LIN {X 0,Y 395.403,Z 549.53,A -85,B 0,C 180,E1 10502.646,E2 10502.646} C_VEL
LIN {X 0,Y 395.709,Z 549.53,A -85,B 0,C 180,E1 10509.858,E2 10509.858} C_VEL
LIN {X 0,Y 395.987,Z 549.53,A -85,B 0,C 180,E1 10516.739,E2 10516.739} C_VEL
LIN {X 0,Y 396.289,Z 549.53,A -85,B 0,C 180,E1 10523.419,E2 10523.419} C_VEL
LIN {X 0,Y 396.65,Z 549.53,A -85,B 0,C 180,E1 10530.001,E2 10530.001} C_VEL
LIN {X 0,Y 396.335,Z 549.53,A -85,B 0,C 180,E1 10536.637,E2 10536.637} C_VEL
LIN {X 0,Y 395.986,Z 549.53,A -85,B 0,C 180,E1 10543.263,E2 10543.263} C_VEL
LIN {X 0,Y 395.756,Z 549.53,A -85,B 0,C 180,E1 10550.141,E2 10550.141} C_VEL
LIN {X 0,Y 395.466,Z 549.53,A -85,B 0,C 180,E1 10557.351,E2 10557.351} C_VEL
LIN {X 0,Y 395.491,Z 550.097,A -85,B 0,C 180,E1 10559.532,E2 10559.532} C_VEL
LIN {X 0,Y 412.664,Z 588.423,A -85,B 0,C 180,E1 10563.55,E2 10563.55} C_VEL
LIN {X 0,Y 423.549,Z 621.01,A -85,B 0,C 180,E1 10567.103,E2 10567.103} C_VEL
LIN {X 0,Y 418.173,Z 655.721,A -85,B 0,C 180,E1 10570.02,E2 10570.02} C_VEL
LIN {X 0,Y 412.096,Z 688.084,A -85,B 0,C 180,E1 10573.717,E2 10573.717} C_VEL
LIN {X 0,Y 406.338,Z 717.384,A -85,B 0,C 180,E1 10578.3,E2 10578.3} C_VEL
LIN {X 0,Y 402.093,Z 739.295,A -85,B 0,C 180,E1 10582.948,E2 10582.948} C_VEL
LIN {X 0,Y 399.09,Z 757.709,A -85,B 0,C 180,E1 10588.375,E2 10588.375} C_VEL
LIN {X 0,Y 397.658,Z 769.165,A -85,B 0,C 180,E1 10593.25,E2 10593.25} C_VEL
LIN {X 0,Y 396.853,Z 777.225,A -85,B 0,C 180,E1 10598.856,E2 10598.856} C_VEL
LIN {X 0,Y 396.449,Z 780.25,A -85,B 0,C 180,E1 10604.49,E2 10604.49} C_VEL
LIN {X 0,Y 396.674,Z 779.113,A -85,B 0,C 180,E1 10608.994,E2 10608.994} C_VEL
LIN {X 0,Y 397.418,Z 773.339,A -85,B 0,C 180,E1 10614.53,E2 10614.53} C_VEL
LIN {X 0,Y 398.697,Z 762.63,A -85,B 0,C 180,E1 10619.995,E2 10619.995} C_VEL
LIN {X 0,Y 401.47,Z 745.337,A -85,B 0,C 180,E1 10625.677,E2 10625.677} C_VEL
LIN {X 0,Y 405.434,Z 724.606,A -85,B 0,C 180,E1 10630.485,E2 10630.485} C_VEL
LIN {X 0,Y 410.682,Z 698.334,A -85,B 0,C 180,E1 10634.951,E2 10634.951} C_VEL
LIN {X 0,Y 416.116,Z 669.777,A -85,B 0,C 180,E1 10638.554,E2 10638.554} C_VEL
LIN {X 0,Y 421.808,Z 635.983,A -85,B 0,C 180,E1 10641.689,E2 10641.689} C_VEL
LIN {X 0,Y 423.501,Z 620.063,A -85,B 0,C 180,E1 10642.925,E2 10642.925} C_VEL
LIN {X 0,Y 412.42,Z 583.384,A -85,B 0,C 180,E1 10646.95,E2 10646.95} C_VEL
LIN {X 0,Y 402.327,Z 561.945,A -85,B 0,C 180,E1 10649.923,E2 10649.923} C_VEL
LIN {X 0,Y 397.745,Z 555.179,A -85,B 0,C 180,E1 10651.335,E2 10651.335} C_VEL
LIN {X 0,Y 395.279,Z 549.53,A -85,B 0,C 180,E1 10652.574,E2 10652.574} C_VEL
LIN {X 0,Y 395.232,Z 549.53,A -85,B 0,C 180,E1 10659.988,E2 10659.988} C_VEL
LIN {X 0,Y 395.279,Z 549.906,A -85,B 0,C 180,E1 10661.254,E2 10661.254} C_VEL
LIN {X 0,Y 397.807,Z 555.344,A -85,B 0,C 180,E1 10662.27,E2 10662.27} C_VEL
LIN {X 0,Y 400.263,Z 559.059,A -85,B 0,C 180,E1 10663.025,E2 10663.025} C_VEL
LIN {X 0,Y 407.693,Z 571.468,A -85,B 0,C 180,E1 10664.926,E2 10664.926} C_VEL
LIN {X 0,Y 418.785,Z 595.422,A -85,B 0,C 180,E1 10667.342,E2 10667.342} C_VEL
LIN {X 0,Y 427.601,Z 621.106,A -85,B 0,C 180,E1 10669.337,E2 10669.337} C_VEL
LIN {X 0,Y 422.708,Z 664.153,A -85,B 0,C 180,E1 10671.265,E2 10671.265} C_VEL
LIN {X 0,Y 417.375,Z 703.599,A -85,B 0,C 180,E1 10673.921,E2 10673.921} C_VEL
LIN {X 0,Y 412.016,Z 738.43,A -85,B 0,C 180,E1 10677.157,E2 10677.157} C_VEL
LIN {X 0,Y 406.992,Z 769.935,A -85,B 0,C 180,E1 10681.077,E2 10681.077} C_VEL
LIN {X 0,Y 404.873,Z 783.295,A -85,B 0,C 180,E1 10683.114,E2 10683.114} C_VEL
LIN {X 0,Y 399.318,Z 794.258,A -85,B 0,C 180,E1 10684.901,E2 10684.901} C_VEL
LIN {X 0,Y 393.912,Z 804.392,A -85,B 0,C 180,E1 10686.826,E2 10686.826} C_VEL
LIN {X 0,Y 391.203,Z 824.838,A -85,B 0,C 180,E1 10691.962,E2 10691.962} C_VEL
LIN {X 0,Y 389.705,Z 839.343,A -85,B 0,C 180,E1 10697.09,E2 10697.09} C_VEL
LIN {X 0,Y 389.124,Z 849,A -85,B 0,C 180,E1 10702.358,E2 10702.358} C_VEL
LIN {X 0,Y 389.002,Z 853.738,A -85,B 0,C 180,E1 10707.768,E2 10707.768} C_VEL
LIN {X 0,Y 389.053,Z 853.851,A -85,B 0,C 180,E1 10712.229,E2 10712.229} C_VEL
LIN {X 0,Y 389.114,Z 849.446,A -85,B 0,C 180,E1 10717.639,E2 10717.639} C_VEL
LIN {X 0,Y 389.754,Z 840.25,A -85,B 0,C 180,E1 10722.906,E2 10722.906} C_VEL
LIN {X 0,Y 391.432,Z 824.911,A -85,B 0,C 180,E1 10728.513,E2 10728.513} C_VEL
LIN {X 0,Y 394.656,Z 803.613,A -85,B 0,C 180,E1 10733.964,E2 10733.964} C_VEL
LIN {X 0,Y 399.5,Z 777.225,A -85,B 0,C 180,E1 10738.894,E2 10738.894} C_VEL
LIN {X 0,Y 405.396,Z 746.474,A -85,B 0,C 180,E1 10743.154,E2 10743.154} C_VEL
LIN {X 0,Y 411.499,Z 713.376,A -85,B 0,C 180,E1 10746.554,E2 10746.554} C_VEL
LIN {X 0,Y 417.568,Z 675.206,A -85,B 0,C 180,E1 10749.384,E2 10749.384} C_VEL
LIN {X 0,Y 422.691,Z 635.88,A -85,B 0,C 180,E1 10751.334,E2 10751.334} C_VEL
LIN {X 0,Y 423.319,Z 622.141,A -85,B 0,C 180,E1 10751.901,E2 10751.901} C_VEL
LIN {X 0,Y 406.224,Z 585.26,A -85,B 0,C 180,E1 10754.989,E2 10754.989} C_VEL
LIN {X 0,Y 387.369,Z 550.77,A -85,B 0,C 180,E1 10758.29,E2 10758.29} C_VEL
LIN {X 0,Y 387.271,Z 549.53,A -85,B 0,C 180,E1 10758.354,E2 10758.354} C_VEL
LIN {X 0,Y 387.319,Z 549.53,A -85,B 0,C 180,E1 10765.174,E2 10765.174} C_VEL
LIN {X 0,Y 387.507,Z 549.53,A -85,B 0,C 180,E1 10772.046,E2 10772.046} C_VEL
LIN {X 0,Y 387.75,Z 549.53,A -85,B 0,C 180,E1 10779.574,E2 10779.574} C_VEL
LIN {X 0,Y 388.026,Z 549.53,A -85,B 0,C 180,E1 10786.466,E2 10786.466} C_VEL
LIN {X 0,Y 388.335,Z 549.53,A -85,B 0,C 180,E1 10793.288,E2 10793.288} C_VEL
LIN {X 0,Y 388.676,Z 549.53,A -85,B 0,C 180,E1 10800.005,E2 10800.005} C_VEL
LIN {X 0,Y 388.415,Z 549.53,A -85,B 0,C 180,E1 10806.72,E2 10806.72} C_VEL
LIN {X 0,Y 388.038,Z 549.53,A -85,B 0,C 180,E1 10813.544,E2 10813.544} C_VEL
LIN {X 0,Y 387.754,Z 549.53,A -85,B 0,C 180,E1 10820.579,E2 10820.579} C_VEL
LIN {X 0,Y 387.504,Z 549.53,A -85,B 0,C 180,E1 10827.965,E2 10827.965} C_VEL
LIN {X 0,Y 387.251,Z 549.53,A -85,B 0,C 180,E1 10835.911,E2 10835.911} C_VEL
LIN {X 0,Y 387.182,Z 549.53,A -85,B 0,C 180,E1 10842.015,E2 10842.015} C_VEL
LIN {X 0,Y 387.146,Z 549.53,A -85,B 0,C 180,E1 10848.331,E2 10848.331} C_VEL
LIN {X 0,Y 387.311,Z 549.53,A -85,B 0,C 180,E1 10855.184,E2 10855.184} C_VEL
LIN {X 0,Y 387.502,Z 549.53,A -85,B 0,C 180,E1 10862.04,E2 10862.04} C_VEL
LIN {X 0,Y 387.775,Z 549.53,A -85,B 0,C 180,E1 10869.576,E2 10869.576} C_VEL
LIN {X 0,Y 388.059,Z 549.53,A -85,B 0,C 180,E1 10876.463,E2 10876.463} C_VEL
LIN {X 0,Y 388.366,Z 549.53,A -85,B 0,C 180,E1 10883.284,E2 10883.284} C_VEL
LIN {X 0,Y 388.755,Z 549.53,A -85,B 0,C 180,E1 10890.001,E2 10890.001} C_VEL
LIN {X 0,Y 388.445,Z 549.53,A -85,B 0,C 180,E1 10896.716,E2 10896.716} C_VEL
LIN {X 0,Y 388.059,Z 549.53,A -85,B 0,C 180,E1 10903.539,E2 10903.539} C_VEL
LIN {X 0,Y 387.784,Z 549.53,A -85,B 0,C 180,E1 10910.574,E2 10910.574} C_VEL
LIN {X 0,Y 387.559,Z 549.53,A -85,B 0,C 180,E1 10918.428,E2 10918.428} C_VEL
LIN {X 0,Y 406.176,Z 591.509,A -85,B 0,C 180,E1 10923.037,E2 10923.037} C_VEL
LIN {X 0,Y 416.831,Z 624.119,A -85,B 0,C 180,E1 10926.704,E2 10926.704} C_VEL
LIN {X 0,Y 410.701,Z 660.444,A -85,B 0,C 180,E1 10929.862,E2 10929.862} C_VEL
LIN {X 0,Y 404.48,Z 691.718,A -85,B 0,C 180,E1 10933.61,E2 10933.61} C_VEL
LIN {X 0,Y 398.9,Z 718.643,A -85,B 0,C 180,E1 10937.967,E2 10937.967} C_VEL
LIN {X 0,Y 394.176,Z 741.909,A -85,B 0,C 180,E1 10943.082,E2 10943.082} C_VEL
LIN {X 0,Y 391.259,Z 759.109,A -85,B 0,C 180,E1 10948.36,E2 10948.36} C_VEL
LIN {X 0,Y 389.678,Z 771.52,A -85,B 0,C 180,E1 10953.988,E2 10953.988} C_VEL
LIN {X 0,Y 388.911,Z 778.598,A -85,B 0,C 180,E1 10959.485,E2 10959.485} C_VEL
LIN {X 0,Y 388.566,Z 780.931,A -85,B 0,C 180,E1 10964.167,E2 10964.167} C_VEL
LIN {X 0,Y 388.787,Z 780.069,A -85,B 0,C 180,E1 10968.767,E2 10968.767} C_VEL
LIN {X 0,Y 389.581,Z 774.519,A -85,B 0,C 180,E1 10974.42,E2 10974.42} C_VEL
LIN {X 0,Y 390.871,Z 764.073,A -85,B 0,C 180,E1 10979.995,E2 10979.995} C_VEL
LIN {X 0,Y 393.623,Z 748.116,A -85,B 0,C 180,E1 10985.513,E2 10985.513} C_VEL
LIN {X 0,Y 397.902,Z 726.736,A -85,B 0,C 180,E1 10990.685,E2 10990.685} C_VEL
LIN {X 0,Y 403.366,Z 700.882,A -85,B 0,C 180,E1 10995.228,E2 10995.228} C_VEL
LIN {X 0,Y 409.287,Z 671.34,A -85,B 0,C 180,E1 10999.06,E2 10999.06} C_VEL
LIN {X 0,Y 415.229,Z 638,A -85,B 0,C 180,E1 11002.224,E2 11002.224} C_VEL
LIN {X 0,Y 417.094,Z 623.357,A -85,B 0,C 180,E1 11003.371,E2 11003.371} C_VEL
LIN {X 0,Y 406.806,Z 587.316,A -85,B 0,C 180,E1 11007.54,E2 11007.54} C_VEL
LIN {X 0,Y 397.957,Z 567.705,A -85,B 0,C 180,E1 11010.474,E2 11010.474} C_VEL
LIN {X 0,Y 391.388,Z 556.424,A -85,B 0,C 180,E1 11013.09,E2 11013.09} C_VEL
LIN {X 0,Y 387.503,Z 551.323,A -85,B 0,C 180,E1 11016.395,E2 11016.395} C_VEL
LIN {X 0,Y 388.184,Z 553.232,A -85,B 0,C 180,E1 11018.548,E2 11018.548} C_VEL
LIN {X 0,Y 392.347,Z 557.901,A -85,B 0,C 180,E1 11020.909,E2 11020.909} C_VEL
LIN {X 0,Y 399.347,Z 569.21,A -85,B 0,C 180,E1 11023.307,E2 11023.307} C_VEL
LIN {X 0,Y 409.854,Z 590.808,A -85,B 0,C 180,E1 11025.985,E2 11025.985} C_VEL
LIN {X 0,Y 420.921,Z 623.838,A -85,B 0,C 180,E1 11028.792,E2 11028.792} C_VEL
LIN {X 0,Y 415.851,Z 665.501,A -85,B 0,C 180,E1 11030.756,E2 11030.756} C_VEL
LIN {X 0,Y 410.134,Z 705.08,A -85,B 0,C 180,E1 11033.516,E2 11033.516} C_VEL
LIN {X 0,Y 404.212,Z 742.136,A -85,B 0,C 180,E1 11037.117,E2 11037.117} C_VEL
LIN {X 0,Y 398.711,Z 774.627,A -85,B 0,C 180,E1 11041.416,E2 11041.416} C_VEL
LIN {X 0,Y 394.369,Z 801.581,A -85,B 0,C 180,E1 11046.226,E2 11046.226} C_VEL
LIN {X 0,Y 393.912,Z 804.392,A -85,B 0,C 180,E1 11046.826,E2 11046.826} C_VEL
LIN {X 0,Y 392.024,Z 809.183,A -85,B 0,C 180,E1 11047.859,E2 11047.859} C_VEL
LIN {X 0,Y 383.939,Z 820.98,A -85,B 0,C 180,E1 11050.755,E2 11050.755} C_VEL
LIN {X 0,Y 383.723,Z 821.96,A -85,B 0,C 180,E1 11051.047,E2 11051.047} C_VEL
LIN {X 0,Y 381.996,Z 837.115,A -85,B 0,C 180,E1 11056.241,E2 11056.241} C_VEL
LIN {X 0,Y 381.365,Z 846.181,A -85,B 0,C 180,E1 11060.861,E2 11060.861} C_VEL
LIN {X 0,Y 381.15,Z 851.589,A -85,B 0,C 180,E1 11065.442,E2 11065.442} C_VEL
LIN {X 0,Y 381.219,Z 853.512,A -85,B 0,C 180,E1 11069.999,E2 11069.999} C_VEL
LIN {X 0,Y 381.128,Z 850.973,A -85,B 0,C 180,E1 11075.699,E2 11075.699} C_VEL
LIN {X 0,Y 381.581,Z 843.003,A -85,B 0,C 180,E1 11081.442,E2 11081.442} C_VEL
LIN {X 0,Y 383.006,Z 829.207,A -85,B 0,C 180,E1 11087.245,E2 11087.245} C_VEL
LIN {X 0,Y 386.095,Z 808.653,A -85,B 0,C 180,E1 11093.087,E2 11093.087} C_VEL
LIN {X 0,Y 390.87,Z 782.989,A -85,B 0,C 180,E1 11098.317,E2 11098.317} C_VEL
LIN {X 0,Y 396.66,Z 754.143,A -85,B 0,C 180,E1 11102.678,E2 11102.678} C_VEL
LIN {X 0,Y 403.169,Z 720.965,A -85,B 0,C 180,E1 11106.401,E2 11106.401} C_VEL
LIN {X 0,Y 409.328,Z 685.638,A -85,B 0,C 180,E1 11109.303,E2 11109.303} C_VEL
LIN {X 0,Y 414.945,Z 647.471,A -85,B 0,C 180,E1 11111.474,E2 11111.474} C_VEL
LIN {X 0,Y 416.878,Z 624.907,A -85,B 0,C 180,E1 11112.446,E2 11112.446} C_VEL
LIN {X 0,Y 399.707,Z 587.708,A -85,B 0,C 180,E1 11115.694,E2 11115.694} C_VEL
LIN {X 0,Y 379.261,Z 550.017,A -85,B 0,C 180,E1 11119.416,E2 11119.416} C_VEL
LIN {X 0,Y 379.445,Z 549.53,A -85,B 0,C 180,E1 11126.922,E2 11126.922} C_VEL
LIN {X 0,Y 379.598,Z 549.53,A -85,B 0,C 180,E1 11133.982,E2 11133.982} C_VEL
LIN {X 0,Y 379.883,Z 549.53,A -85,B 0,C 180,E1 11141.412,E2 11141.412} C_VEL
LIN {X 0,Y 380.175,Z 549.53,A -85,B 0,C 180,E1 11148.519,E2 11148.519} C_VEL
LIN {X 0,Y 380.544,Z 549.53,A -85,B 0,C 180,E1 11155.441,E2 11155.441} C_VEL
LIN {X 0,Y 380.805,Z 549.53,A -85,B 0,C 180,E1 11162.283,E2 11162.283} C_VEL
LIN {X 0,Y 380.312,Z 549.53,A -85,B 0,C 180,E1 11169.168,E2 11169.168} C_VEL
LIN {X 0,Y 379.993,Z 549.53,A -85,B 0,C 180,E1 11176.2,E2 11176.2} C_VEL
LIN {X 0,Y 379.691,Z 549.53,A -85,B 0,C 180,E1 11183.505,E2 11183.505} C_VEL
LIN {X 0,Y 379.522,Z 549.53,A -85,B 0,C 180,E1 11188.64,E2 11188.64} C_VEL
LIN {X 0,Y 379.353,Z 549.53,A -85,B 0,C 180,E1 11193.975,E2 11193.975} C_VEL
LIN {X 0,Y 379.199,Z 549.53,A -85,B 0,C 180,E1 11200.658,E2 11200.658} C_VEL
LIN {X 0,Y 379.163,Z 549.53,A -85,B 0,C 180,E1 11207.248,E2 11207.248} C_VEL
LIN {X 0,Y 379.259,Z 549.53,A -85,B 0,C 180,E1 11213.215,E2 11213.215} C_VEL
LIN {X 0,Y 379.424,Z 549.53,A -85,B 0,C 180,E1 11218.752,E2 11218.752} C_VEL
LIN {X 0,Y 379.651,Z 549.53,A -85,B 0,C 180,E1 11226.498,E2 11226.498} C_VEL
LIN {X 0,Y 380.009,Z 549.53,A -85,B 0,C 180,E1 11233.806,E2 11233.806} C_VEL
LIN {X 0,Y 380.345,Z 549.53,A -85,B 0,C 180,E1 11240.839,E2 11240.839} C_VEL
LIN {X 0,Y 380.768,Z 549.53,A -85,B 0,C 180,E1 11247.722,E2 11247.722} C_VEL
LIN {X 0,Y 380.544,Z 549.53,A -85,B 0,C 180,E1 11254.565,E2 11254.565} C_VEL
LIN {X 0,Y 380.178,Z 549.53,A -85,B 0,C 180,E1 11261.487,E2 11261.487} C_VEL
LIN {X 0,Y 379.933,Z 549.53,A -85,B 0,C 180,E1 11268.592,E2 11268.592} C_VEL
LIN {X 0,Y 379.667,Z 549.53,A -85,B 0,C 180,E1 11276.02,E2 11276.02} C_VEL
LIN {X 0,Y 379.62,Z 549.767,A -85,B 0,C 180,E1 11277.463,E2 11277.463} C_VEL
LIN {X 0,Y 396.65,Z 587.157,A -85,B 0,C 180,E1 11281.66,E2 11281.66} C_VEL
LIN {X 0,Y 407.431,Z 617.515,A -85,B 0,C 180,E1 11285.154,E2 11285.154} C_VEL
LIN {X 0,Y 409.836,Z 628.295,A -85,B 0,C 180,E1 11286.371,E2 11286.371} C_VEL
LIN {X 0,Y 403.587,Z 662.712,A -85,B 0,C 180,E1 11289.471,E2 11289.471} C_VEL
LIN {X 0,Y 397.063,Z 694.134,A -85,B 0,C 180,E1 11293.345,E2 11293.345} C_VEL
LIN {X 0,Y 391.503,Z 719.773,A -85,B 0,C 180,E1 11297.596,E2 11297.596} C_VEL
LIN {X 0,Y 386.689,Z 742.384,A -85,B 0,C 180,E1 11302.652,E2 11302.652} C_VEL
LIN {X 0,Y 383.785,Z 758.729,A -85,B 0,C 180,E1 11307.669,E2 11307.669} C_VEL
LIN {X 0,Y 381.954,Z 771.588,A -85,B 0,C 180,E1 11313.422,E2 11313.422} C_VEL
LIN {X 0,Y 381.129,Z 779.042,A -85,B 0,C 180,E1 11319.047,E2 11319.047} C_VEL
LIN {X 0,Y 380.695,Z 781.607,A -85,B 0,C 180,E1 11323.831,E2 11323.831} C_VEL
LIN {X 0,Y 380.905,Z 780.952,A -85,B 0,C 180,E1 11328.532,E2 11328.532} C_VEL
LIN {X 0,Y 381.725,Z 775.68,A -85,B 0,C 180,E1 11334.305,E2 11334.305} C_VEL
LIN {X 0,Y 383.074,Z 765.499,A -85,B 0,C 180,E1 11339.995,E2 11339.995} C_VEL
LIN {X 0,Y 385.914,Z 749.858,A -85,B 0,C 180,E1 11345.624,E2 11345.624} C_VEL
LIN {X 0,Y 390.657,Z 727.583,A -85,B 0,C 180,E1 11351.169,E2 11351.169} C_VEL
LIN {X 0,Y 396.455,Z 701.727,A -85,B 0,C 180,E1 11355.784,E2 11355.784} C_VEL
LIN {X 0,Y 402.57,Z 672.766,A -85,B 0,C 180,E1 11359.607,E2 11359.607} C_VEL
LIN {X 0,Y 408.78,Z 639.82,A -85,B 0,C 180,E1 11362.801,E2 11362.801} C_VEL
LIN {X 0,Y 410.607,Z 625.996,A -85,B 0,C 180,E1 11363.924,E2 11363.924} C_VEL
LIN {X 0,Y 401.362,Z 591.182,A -85,B 0,C 180,E1 11368.161,E2 11368.161} C_VEL
LIN {X 0,Y 393.451,Z 572.822,A -85,B 0,C 180,E1 11371.155,E2 11371.155} C_VEL
LIN {X 0,Y 388.4,Z 563.472,A -85,B 0,C 180,E1 11373.572,E2 11373.572} C_VEL
LIN {X 0,Y 385.702,Z 558.895,A -85,B 0,C 180,E1 11376.643,E2 11376.643} C_VEL
LIN {X 0,Y 387.625,Z 562.694,A -85,B 0,C 180,E1 11379.483,E2 11379.483} C_VEL
LIN {X 0,Y 389.867,Z 565.725,A -85,B 0,C 180,E1 11380.663,E2 11380.663} C_VEL
LIN {X 0,Y 396.008,Z 576.315,A -85,B 0,C 180,E1 11382.965,E2 11382.965} C_VEL
LIN {X 0,Y 405.521,Z 597.346,A -85,B 0,C 180,E1 11385.653,E2 11385.653} C_VEL
LIN {X 0,Y 414.457,Z 626.276,A -85,B 0,C 180,E1 11388.219,E2 11388.219} C_VEL
LIN {X 0,Y 408.852,Z 668.458,A -85,B 0,C 180,E1 11390.314,E2 11390.314} C_VEL
LIN {X 0,Y 402.463,Z 709.436,A -85,B 0,C 180,E1 11393.333,E2 11393.333} C_VEL
LIN {X 0,Y 396.386,Z 745.076,A -85,B 0,C 180,E1 11397.003,E2 11397.003} C_VEL
LIN {X 0,Y 391.015,Z 775.388,A -85,B 0,C 180,E1 11401.188,E2 11401.188} C_VEL
LIN {X 0,Y 386.608,Z 801.678,A -85,B 0,C 180,E1 11406.025,E2 11406.025} C_VEL
LIN {X 0,Y 383.723,Z 821.96,A -85,B 0,C 180,E1 11411.047,E2 11411.047} C_VEL
LIN {X 0,Y 380.541,Z 827.599,A -85,B 0,C 180,E1 11412.77,E2 11412.77} C_VEL
LIN {X 0,Y 374.405,Z 834.833,A -85,B 0,C 180,E1 11415.415,E2 11415.415} C_VEL
LIN {X 0,Y 374.233,Z 835.617,A -85,B 0,C 180,E1 11415.728,E2 11415.728} C_VEL
LIN {X 0,Y 373.5,Z 845.344,A -85,B 0,C 180,E1 11420.667,E2 11420.667} C_VEL
LIN {X 0,Y 373.272,Z 850.797,A -85,B 0,C 180,E1 11425.346,E2 11425.346} C_VEL
LIN {X 0,Y 373.37,Z 852.773,A -85,B 0,C 180,E1 11429.999,E2 11429.999} C_VEL
LIN {X 0,Y 373.266,Z 850.397,A -85,B 0,C 180,E1 11435.627,E2 11435.627} C_VEL
LIN {X 0,Y 373.676,Z 843.277,A -85,B 0,C 180,E1 11441.095,E2 11441.095} C_VEL
LIN {X 0,Y 374.794,Z 831.64,A -85,B 0,C 180,E1 11446.425,E2 11446.425} C_VEL
LIN {X 0,Y 377.464,Z 813.611,A -85,B 0,C 180,E1 11452.074,E2 11452.074} C_VEL
LIN {X 0,Y 381.896,Z 790.449,A -85,B 0,C 180,E1 11457.317,E2 11457.317} C_VEL
LIN {X 0,Y 387.58,Z 762.592,A -85,B 0,C 180,E1 11461.992,E2 11461.992} C_VEL
LIN {X 0,Y 393.997,Z 731.725,A -85,B 0,C 180,E1 11465.862,E2 11465.862} C_VEL
LIN {X 0,Y 400.746,Z 697.058,A -85,B 0,C 180,E1 11469.062,E2 11469.062} C_VEL
LIN {X 0,Y 406.674,Z 660.675,A -85,B 0,C 180,E1 11471.452,E2 11471.452} C_VEL
LIN {X 0,Y 410.203,Z 627.23,A -85,B 0,C 180,E1 11473.036,E2 11473.036} C_VEL
LIN {X 0,Y 393.747,Z 591.126,A -85,B 0,C 180,E1 11476.303,E2 11476.303} C_VEL
LIN {X 0,Y 371.419,Z 550.834,A -85,B 0,C 180,E1 11480.496,E2 11480.496} C_VEL
LIN {X 0,Y 371.29,Z 549.53,A -85,B 0,C 180,E1 11480.785,E2 11480.785} C_VEL
LIN {X 0,Y 371.497,Z 549.53,A -85,B 0,C 180,E1 11488.013,E2 11488.013} C_VEL
LIN {X 0,Y 371.67,Z 549.53,A -85,B 0,C 180,E1 11495.966,E2 11495.966} C_VEL
LIN {X 0,Y 372.061,Z 549.53,A -85,B 0,C 180,E1 11503.455,E2 11503.455} C_VEL
LIN {X 0,Y 372.378,Z 549.53,A -85,B 0,C 180,E1 11510.645,E2 11510.645} C_VEL
LIN {X 0,Y 372.782,Z 549.53,A -85,B 0,C 180,E1 11517.677,E2 11517.677} C_VEL
LIN {X 0,Y 372.888,Z 549.53,A -85,B 0,C 180,E1 11522.332,E2 11522.332} C_VEL
LIN {X 0,Y 372.373,Z 549.53,A -85,B 0,C 180,E1 11529.365,E2 11529.365} C_VEL
LIN {X 0,Y 372.071,Z 549.53,A -85,B 0,C 180,E1 11536.555,E2 11536.555} C_VEL
LIN {X 0,Y 371.714,Z 549.53,A -85,B 0,C 180,E1 11544.041,E2 11544.041} C_VEL
LIN {X 0,Y 371.492,Z 549.53,A -85,B 0,C 180,E1 11551.145,E2 11551.145} C_VEL
LIN {X 0,Y 371.263,Z 549.53,A -85,B 0,C 180,E1 11557.719,E2 11557.719} C_VEL
LIN {X 0,Y 371.274,Z 549.53,A -85,B 0,C 180,E1 11563.894,E2 11563.894} C_VEL
LIN {X 0,Y 371.256,Z 549.53,A -85,B 0,C 180,E1 11570.798,E2 11570.798} C_VEL
LIN {X 0,Y 371.498,Z 549.53,A -85,B 0,C 180,E1 11578.008,E2 11578.008} C_VEL
LIN {X 0,Y 371.68,Z 549.53,A -85,B 0,C 180,E1 11585.962,E2 11585.962} C_VEL
LIN {X 0,Y 372.085,Z 549.53,A -85,B 0,C 180,E1 11593.452,E2 11593.452} C_VEL
LIN {X 0,Y 372.407,Z 549.53,A -85,B 0,C 180,E1 11600.642,E2 11600.642} C_VEL
LIN {X 0,Y 372.859,Z 549.53,A -85,B 0,C 180,E1 11607.674,E2 11607.674} C_VEL
LIN {X 0,Y 372.895,Z 549.53,A -85,B 0,C 180,E1 11612.328,E2 11612.328} C_VEL
LIN {X 0,Y 372.394,Z 549.53,A -85,B 0,C 180,E1 11619.361,E2 11619.361} C_VEL
LIN {X 0,Y 372.101,Z 549.53,A -85,B 0,C 180,E1 11626.55,E2 11626.55} C_VEL
LIN {X 0,Y 371.741,Z 549.53,A -85,B 0,C 180,E1 11634.036,E2 11634.036} C_VEL
LIN {X 0,Y 371.743,Z 549.53,A -85,B 0,C 180,E1 11636.351,E2 11636.351} C_VEL
LIN {X 0,Y 378.606,Z 564.621,A -85,B 0,C 180,E1 11638.047,E2 11638.047} C_VEL
LIN {X 0,Y 393.249,Z 597.892,A -85,B 0,C 180,E1 11642.009,E2 11642.009} C_VEL
LIN {X 0,Y 403.104,Z 629.27,A -85,B 0,C 180,E1 11645.756,E2 11645.756} C_VEL
LIN {X 0,Y 396.611,Z 664.345,A -85,B 0,C 180,E1 11648.995,E2 11648.995} C_VEL
LIN {X 0,Y 390.002,Z 694.877,A -85,B 0,C 180,E1 11652.829,E2 11652.829} C_VEL
LIN {X 0,Y 383.799,Z 722.207,A -85,B 0,C 180,E1 11657.478,E2 11657.478} C_VEL
LIN {X 0,Y 378.993,Z 743.931,A -85,B 0,C 180,E1 11662.5,E2 11662.5} C_VEL
LIN {X 0,Y 375.887,Z 760.449,A -85,B 0,C 180,E1 11667.768,E2 11667.768} C_VEL
LIN {X 0,Y 374.094,Z 772.834,A -85,B 0,C 180,E1 11673.559,E2 11673.559} C_VEL
LIN {X 0,Y 373.297,Z 779.703,A -85,B 0,C 180,E1 11678.888,E2 11678.888} C_VEL
LIN {X 0,Y 372.831,Z 782.285,A -85,B 0,C 180,E1 11683.48,E2 11683.48} C_VEL
LIN {X 0,Y 373.012,Z 781.841,A -85,B 0,C 180,E1 11688.286,E2 11688.286} C_VEL
LIN {X 0,Y 373.875,Z 776.824,A -85,B 0,C 180,E1 11694.201,E2 11694.201} C_VEL
LIN {X 0,Y 375.255,Z 766.962,A -85,B 0,C 180,E1 11699.995,E2 11699.995} C_VEL
LIN {X 0,Y 378.203,Z 751.625,A -85,B 0,C 180,E1 11705.739,E2 11705.739} C_VEL
LIN {X 0,Y 382.884,Z 731.039,A -85,B 0,C 180,E1 11711.11,E2 11711.11} C_VEL
LIN {X 0,Y 389.218,Z 704.427,A -85,B 0,C 180,E1 11716.086,E2 11716.086} C_VEL
LIN {X 0,Y 395.834,Z 674.708,A -85,B 0,C 180,E1 11720.131,E2 11720.131} C_VEL
LIN {X 0,Y 402.412,Z 641.64,A -85,B 0,C 180,E1 11723.411,E2 11723.411} C_VEL
LIN {X 0,Y 404.066,Z 628.441,A -85,B 0,C 180,E1 11724.548,E2 11724.548} C_VEL
LIN {X 0,Y 395.849,Z 594.745,A -85,B 0,C 180,E1 11728.865,E2 11728.865} C_VEL
LIN {X 0,Y 388.533,Z 576.11,A -85,B 0,C 180,E1 11732.212,E2 11732.212} C_VEL
LIN {X 0,Y 385.348,Z 570.356,A -85,B 0,C 180,E1 11734.106,E2 11734.106} C_VEL
LIN {X 0,Y 383.822,Z 566.965,A -85,B 0,C 180,E1 11736.271,E2 11736.271} C_VEL
LIN {X 0,Y 384.156,Z 568.14,A -85,B 0,C 180,E1 11738.086,E2 11738.086} C_VEL
LIN {X 0,Y 387.053,Z 572.668,A -85,B 0,C 180,E1 11740.267,E2 11740.267} C_VEL
LIN {X 0,Y 392.786,Z 583.519,A -85,B 0,C 180,E1 11742.643,E2 11742.643} C_VEL
LIN {X 0,Y 401.104,Z 603.996,A -85,B 0,C 180,E1 11745.317,E2 11745.317} C_VEL
LIN {X 0,Y 407.947,Z 629.582,A -85,B 0,C 180,E1 11747.645,E2 11747.645} C_VEL
LIN {X 0,Y 401.622,Z 673.297,A -85,B 0,C 180,E1 11749.982,E2 11749.982} C_VEL
LIN {X 0,Y 394.93,Z 712.853,A -85,B 0,C 180,E1 11753.08,E2 11753.08} C_VEL
LIN {X 0,Y 388.777,Z 746.941,A -85,B 0,C 180,E1 11756.753,E2 11756.753} C_VEL
LIN {X 0,Y 383.024,Z 778.032,A -85,B 0,C 180,E1 11761.245,E2 11761.245} C_VEL
LIN {X 0,Y 378.352,Z 804.531,A -85,B 0,C 180,E1 11766.41,E2 11766.41} C_VEL
LIN {X 0,Y 375.476,Z 824.667,A -85,B 0,C 180,E1 11771.788,E2 11771.788} C_VEL
LIN {X 0,Y 374.233,Z 835.617,A -85,B 0,C 180,E1 11775.728,E2 11775.728} C_VEL
LIN {X 0,Y 371.371,Z 839.752,A -85,B 0,C 180,E1 11777.594,E2 11777.594} C_VEL
LIN {X 0,Y 365.604,Z 845,A -85,B 0,C 180,E1 11780.807,E2 11780.807} C_VEL
LIN {X 0,Y 365.394,Z 850.021,A -85,B 0,C 180,E1 11785.245,E2 11785.245} C_VEL
LIN {X 0,Y 365.522,Z 852.031,A -85,B 0,C 180,E1 11789.999,E2 11789.999} C_VEL
LIN {X 0,Y 365.354,Z 850.408,A -85,B 0,C 180,E1 11794.753,E2 11794.753} C_VEL
LIN {X 0,Y 365.762,Z 843.535,A -85,B 0,C 180,E1 11800.735,E2 11800.735} C_VEL
LIN {X 0,Y 366.845,Z 832.426,A -85,B 0,C 180,E1 11806.175,E2 11806.175} C_VEL
LIN {X 0,Y 369.54,Z 814.548,A -85,B 0,C 180,E1 11812.063,E2 11812.063} C_VEL
LIN {X 0,Y 374.177,Z 791.131,A -85,B 0,C 180,E1 11817.55,E2 11817.55} C_VEL
LIN {X 0,Y 380.12,Z 763.354,A -85,B 0,C 180,E1 11822.358,E2 11822.358} C_VEL
LIN {X 0,Y 386.911,Z 732.115,A -85,B 0,C 180,E1 11826.374,E2 11826.374} C_VEL
LIN {X 0,Y 394.173,Z 695.949,A -85,B 0,C 180,E1 11829.755,E2 11829.755} C_VEL
LIN {X 0,Y 400.543,Z 658.231,A -85,B 0,C 180,E1 11832.231,E2 11832.231} C_VEL
LIN {X 0,Y 403.786,Z 630.204,A -85,B 0,C 180,E1 11833.571,E2 11833.571} C_VEL
LIN {X 0,Y 388.137,Z 595.327,A -85,B 0,C 180,E1 11836.861,E2 11836.861} C_VEL
LIN {X 0,Y 363.449,Z 550.644,A -85,B 0,C 180,E1 11841.682,E2 11841.682} C_VEL
LIN {X 0,Y 363.353,Z 549.53,A -85,B 0,C 180,E1 11841.877,E2 11841.877} C_VEL
LIN {X 0,Y 363.469,Z 549.53,A -85,B 0,C 180,E1 11847.219,E2 11847.219} C_VEL
LIN {X 0,Y 363.624,Z 549.53,A -85,B 0,C 180,E1 11852.747,E2 11852.747} C_VEL
LIN {X 0,Y 363.984,Z 549.53,A -85,B 0,C 180,E1 11860.568,E2 11860.568} C_VEL
LIN {X 0,Y 364.315,Z 549.53,A -85,B 0,C 180,E1 11868.012,E2 11868.012} C_VEL
LIN {X 0,Y 364.727,Z 549.53,A -85,B 0,C 180,E1 11875.243,E2 11875.243} C_VEL
LIN {X 0,Y 364.972,Z 549.53,A -85,B 0,C 180,E1 11882.382,E2 11882.382} C_VEL
LIN {X 0,Y 364.432,Z 549.53,A -85,B 0,C 180,E1 11889.571,E2 11889.571} C_VEL
LIN {X 0,Y 364.12,Z 549.53,A -85,B 0,C 180,E1 11896.99,E2 11896.99} C_VEL
LIN {X 0,Y 363.758,Z 549.53,A -85,B 0,C 180,E1 11904.602,E2 11904.602} C_VEL
LIN {X 0,Y 363.605,Z 549.53,A -85,B 0,C 180,E1 11909.984,E2 11909.984} C_VEL
LIN {X 0,Y 363.376,Z 549.53,A -85,B 0,C 180,E1 11917.66,E2 11917.66} C_VEL
LIN {X 0,Y 363.318,Z 549.53,A -85,B 0,C 180,E1 11924.893,E2 11924.893} C_VEL
LIN {X 0,Y 363.366,Z 549.53,A -85,B 0,C 180,E1 11932.35,E2 11932.35} C_VEL
LIN {X 0,Y 363.613,Z 549.53,A -85,B 0,C 180,E1 11940.023,E2 11940.023} C_VEL
LIN {X 0,Y 363.819,Z 549.53,A -85,B 0,C 180,E1 11948.005,E2 11948.005} C_VEL
LIN {X 0,Y 364.218,Z 549.53,A -85,B 0,C 180,E1 11955.558,E2 11955.558} C_VEL
LIN {X 0,Y 364.605,Z 549.53,A -85,B 0,C 180,E1 11962.845,E2 11962.845} C_VEL
LIN {X 0,Y 365.051,Z 549.53,A -85,B 0,C 180,E1 11970.001,E2 11970.001} C_VEL
LIN {X 0,Y 364.692,Z 549.53,A -85,B 0,C 180,E1 11977.156,E2 11977.156} C_VEL
LIN {X 0,Y 364.222,Z 549.53,A -85,B 0,C 180,E1 11984.444,E2 11984.444} C_VEL
LIN {X 0,Y 363.868,Z 549.53,A -85,B 0,C 180,E1 11991.994,E2 11991.994} C_VEL
LIN {X 0,Y 363.786,Z 549.797,A -85,B 0,C 180,E1 11995.232,E2 11995.232} C_VEL
LIN {X 0,Y 373.547,Z 570.156,A -85,B 0,C 180,E1 11997.676,E2 11997.676} C_VEL
LIN {X 0,Y 388.204,Z 605.005,A -85,B 0,C 180,E1 12001.952,E2 12001.952} C_VEL
LIN {X 0,Y 396.284,Z 631.972,A -85,B 0,C 180,E1 12005.302,E2 12005.302} C_VEL
LIN {X 0,Y 389.491,Z 666.717,A -85,B 0,C 180,E1 12008.59,E2 12008.59} C_VEL
LIN {X 0,Y 382.588,Z 697.257,A -85,B 0,C 180,E1 12012.541,E2 12012.541} C_VEL
LIN {X 0,Y 376.309,Z 723.715,A -85,B 0,C 180,E1 12017.173,E2 12017.173} C_VEL
LIN {X 0,Y 371.351,Z 745.268,A -85,B 0,C 180,E1 12022.291,E2 12022.291} C_VEL
LIN {X 0,Y 368.103,Z 761.66,A -85,B 0,C 180,E1 12027.671,E2 12027.671} C_VEL
LIN {X 0,Y 366.229,Z 773.925,A -85,B 0,C 180,E1 12033.609,E2 12033.609} C_VEL
LIN {X 0,Y 365.303,Z 781.03,A -85,B 0,C 180,E1 12039.595,E2 12039.595} C_VEL
LIN {X 0,Y 364.98,Z 783.235,A -85,B 0,C 180,E1 12045.583,E2 12045.583} C_VEL
LIN {X 0,Y 365.548,Z 780.502,A -85,B 0,C 180,E1 12051.66,E2 12051.66} C_VEL
LIN {X 0,Y 366.728,Z 772.905,A -85,B 0,C 180,E1 12057.629,E2 12057.629} C_VEL
LIN {X 0,Y 369.079,Z 760.143,A -85,B 0,C 180,E1 12063.523,E2 12063.523} C_VEL
LIN {X 0,Y 373.297,Z 741.432,A -85,B 0,C 180,E1 12069.332,E2 12069.332} C_VEL
LIN {X 0,Y 379.13,Z 718.206,A -85,B 0,C 180,E1 12074.448,E2 12074.448} C_VEL
LIN {X 0,Y 385.871,Z 690.699,A -85,B 0,C 180,E1 12078.882,E2 12078.882} C_VEL
LIN {X 0,Y 393.145,Z 658.726,A -85,B 0,C 180,E1 12082.645,E2 12082.645} C_VEL
LIN {X 0,Y 397.868,Z 631.854,A -85,B 0,C 180,E1 12085.078,E2 12085.078} C_VEL
LIN {X 0,Y 390.753,Z 599.088,A -85,B 0,C 180,E1 12089.493,E2 12089.493} C_VEL
LIN {X 0,Y 384.866,Z 582.333,A -85,B 0,C 180,E1 12092.751,E2 12092.751} C_VEL
LIN {X 0,Y 382.538,Z 577.334,A -85,B 0,C 180,E1 12094.587,E2 12094.587} C_VEL
LIN {X 0,Y 381.866,Z 574.457,A -85,B 0,C 180,E1 12097.072,E2 12097.072} C_VEL
LIN {X 0,Y 384.391,Z 579.833,A -85,B 0,C 180,E1 12099.918,E2 12099.918} C_VEL
LIN {X 0,Y 389.565,Z 590.854,A -85,B 0,C 180,E1 12102.399,E2 12102.399} C_VEL
LIN {X 0,Y 397.24,Z 612.814,A -85,B 0,C 180,E1 12105.217,E2 12105.217} C_VEL
LIN {X 0,Y 401.72,Z 631.423,A -85,B 0,C 180,E1 12106.992,E2 12106.992} C_VEL
LIN {X 0,Y 395.099,Z 673.808,A -85,B 0,C 180,E1 12109.347,E2 12109.347} C_VEL
LIN {X 0,Y 388.119,Z 712.679,A -85,B 0,C 180,E1 12112.471,E2 12112.471} C_VEL
LIN {X 0,Y 381.377,Z 748.024,A -85,B 0,C 180,E1 12116.384,E2 12116.384} C_VEL
LIN {X 0,Y 375.295,Z 779.149,A -85,B 0,C 180,E1 12121.044,E2 12121.044} C_VEL
LIN {X 0,Y 370.469,Z 805.258,A -85,B 0,C 180,E1 12126.336,E2 12126.336} C_VEL
LIN {X 0,Y 367.616,Z 824.588,A -85,B 0,C 180,E1 12131.687,E2 12131.687} C_VEL
LIN {X 0,Y 366.056,Z 838.399,A -85,B 0,C 180,E1 12137.091,E2 12137.091} C_VEL
LIN {X 0,Y 365.604,Z 845,A -85,B 0,C 180,E1 12140.807,E2 12140.807} C_VEL
LIN {X 0,Y 364.225,Z 846.756,A -85,B 0,C 180,E1 12142.136,E2 12142.136} C_VEL
LIN {X 0,Y 357.475,Z 849.916,A -85,B 0,C 180,E1 12146.087,E2 12146.087} C_VEL
LIN {X 0,Y 357.468,Z 849.861,A -85,B 0,C 180,E1 12146.174,E2 12146.174} C_VEL
LIN {X 0,Y 357.666,Z 851.288,A -85,B 0,C 180,E1 12149.999,E2 12149.999} C_VEL
LIN {X 0,Y 357.501,Z 849.671,A -85,B 0,C 180,E1 12154.858,E2 12154.858} C_VEL
LIN {X 0,Y 357.883,Z 842.769,A -85,B 0,C 180,E1 12160.974,E2 12160.974} C_VEL
LIN {X 0,Y 359.04,Z 831.603,A -85,B 0,C 180,E1 12166.537,E2 12166.537} C_VEL
LIN {X 0,Y 362.075,Z 813.067,A -85,B 0,C 180,E1 12172.687,E2 12172.687} C_VEL
LIN {X 0,Y 367.032,Z 789.176,A -85,B 0,C 180,E1 12178.319,E2 12178.319} C_VEL
LIN {X 0,Y 373.292,Z 761.333,A -85,B 0,C 180,E1 12183.144,E2 12183.144} C_VEL
LIN {X 0,Y 380.612,Z 728.825,A -85,B 0,C 180,E1 12187.298,E2 12187.298} C_VEL
LIN {X 0,Y 388.275,Z 691.783,A -85,B 0,C 180,E1 12190.714,E2 12190.714} C_VEL
LIN {X 0,Y 395.109,Z 652.042,A -85,B 0,C 180,E1 12193.227,E2 12193.227} C_VEL
LIN {X 0,Y 397.026,Z 632.119,A -85,B 0,C 180,E1 12194.212,E2 12194.212} C_VEL
LIN {X 0,Y 380.793,Z 596.117,A -85,B 0,C 180,E1 12197.77,E2 12197.77} C_VEL
LIN {X 0,Y 355.523,Z 550.708,A -85,B 0,C 180,E1 12202.9,E2 12202.9} C_VEL
LIN {X 0,Y 355.437,Z 549.53,A -85,B 0,C 180,E1 12203.144,E2 12203.144} C_VEL
LIN {X 0,Y 355.595,Z 549.53,A -85,B 0,C 180,E1 12209.28,E2 12209.28} C_VEL
LIN {X 0,Y 355.732,Z 549.53,A -85,B 0,C 180,E1 12214.816,E2 12214.816} C_VEL
LIN {X 0,Y 356.171,Z 549.53,A -85,B 0,C 180,E1 12222.694,E2 12222.694} C_VEL
LIN {X 0,Y 356.5,Z 549.53,A -85,B 0,C 180,E1 12230.225,E2 12230.225} C_VEL
LIN {X 0,Y 356.965,Z 549.53,A -85,B 0,C 180,E1 12237.574,E2 12237.574} C_VEL
LIN {X 0,Y 357.084,Z 549.53,A -85,B 0,C 180,E1 12242.435,E2 12242.435} C_VEL
LIN {X 0,Y 356.492,Z 549.53,A -85,B 0,C 180,E1 12249.786,E2 12249.786} C_VEL
LIN {X 0,Y 356.191,Z 549.53,A -85,B 0,C 180,E1 12257.315,E2 12257.315} C_VEL
LIN {X 0,Y 355.763,Z 549.53,A -85,B 0,C 180,E1 12265.192,E2 12265.192} C_VEL
LIN {X 0,Y 355.502,Z 549.53,A -85,B 0,C 180,E1 12271.595,E2 12271.595} C_VEL
LIN {X 0,Y 355.438,Z 549.53,A -85,B 0,C 180,E1 12276.615,E2 12276.615} C_VEL
LIN {X 0,Y 355.316,Z 549.53,A -85,B 0,C 180,E1 12283.582,E2 12283.582} C_VEL
LIN {X 0,Y 355.353,Z 549.53,A -85,B 0,C 180,E1 12290.276,E2 12290.276} C_VEL
LIN {X 0,Y 355.507,Z 549.53,A -85,B 0,C 180,E1 12296.383,E2 12296.383} C_VEL
LIN {X 0,Y 355.714,Z 549.53,A -85,B 0,C 180,E1 12303.369,E2 12303.369} C_VEL
LIN {X 0,Y 356.025,Z 549.53,A -85,B 0,C 180,E1 12310.111,E2 12310.111} C_VEL
LIN {X 0,Y 356.412,Z 549.53,A -85,B 0,C 180,E1 12317.738,E2 12317.738} C_VEL
LIN {X 0,Y 356.932,Z 549.53,A -85,B 0,C 180,E1 12325.134,E2 12325.134} C_VEL
LIN {X 0,Y 357.091,Z 549.53,A -85,B 0,C 180,E1 12332.431,E2 12332.431} C_VEL
LIN {X 0,Y 356.514,Z 549.53,A -85,B 0,C 180,E1 12339.782,E2 12339.782} C_VEL
LIN {X 0,Y 356.213,Z 549.53,A -85,B 0,C 180,E1 12347.31,E2 12347.31} C_VEL
LIN {X 0,Y 355.908,Z 549.614,A -85,B 0,C 180,E1 12354.045,E2 12354.045} C_VEL
LIN {X 0,Y 360.496,Z 559.885,A -85,B 0,C 180,E1 12355.25,E2 12355.25} C_VEL
LIN {X 0,Y 376.506,Z 594.418,A -85,B 0,C 180,E1 12359.679,E2 12359.679} C_VEL
LIN {X 0,Y 387.222,Z 625.776,A -85,B 0,C 180,E1 12363.678,E2 12363.678} C_VEL
LIN {X 0,Y 389.141,Z 636.065,A -85,B 0,C 180,E1 12364.936,E2 12364.936} C_VEL
LIN {X 0,Y 381.862,Z 671.195,A -85,B 0,C 180,E1 12368.413,E2 12368.413} C_VEL
LIN {X 0,Y 374.463,Z 702.631,A -85,B 0,C 180,E1 12372.716,E2 12372.716} C_VEL
LIN {X 0,Y 368.134,Z 728.098,A -85,B 0,C 180,E1 12377.462,E2 12377.462} C_VEL
LIN {X 0,Y 363.141,Z 749.029,A -85,B 0,C 180,E1 12382.773,E2 12382.773} C_VEL
LIN {X 0,Y 359.93,Z 764.863,A -85,B 0,C 180,E1 12388.378,E2 12388.378} C_VEL
LIN {X 0,Y 358.356,Z 775.094,A -85,B 0,C 180,E1 12393.712,E2 12393.712} C_VEL
LIN {X 0,Y 357.532,Z 781.148,A -85,B 0,C 180,E1 12398.696,E2 12398.696} C_VEL
LIN {X 0,Y 357.088,Z 784.019,A -85,B 0,C 180,E1 12405.257,E2 12405.257} C_VEL
LIN {X 0,Y 357.655,Z 781.368,A -85,B 0,C 180,E1 12411.593,E2 12411.593} C_VEL
LIN {X 0,Y 358.898,Z 774.291,A -85,B 0,C 180,E1 12417.577,E2 12417.577} C_VEL
LIN {X 0,Y 361.356,Z 761.85,A -85,B 0,C 180,E1 12423.598,E2 12423.598} C_VEL
LIN {X 0,Y 365.734,Z 743.504,A -85,B 0,C 180,E1 12429.526,E2 12429.526} C_VEL
LIN {X 0,Y 371.791,Z 720.722,A -85,B 0,C 180,E1 12434.74,E2 12434.74} C_VEL
LIN {X 0,Y 378.809,Z 693.808,A -85,B 0,C 180,E1 12439.248,E2 12439.248} C_VEL
LIN {X 0,Y 386.304,Z 662.657,A -85,B 0,C 180,E1 12443.069,E2 12443.069} C_VEL
LIN {X 0,Y 391.739,Z 634.83,A -85,B 0,C 180,E1 12445.693,E2 12445.693} C_VEL
LIN {X 0,Y 385.677,Z 602.731,A -85,B 0,C 180,E1 12450.268,E2 12450.268} C_VEL
LIN {X 0,Y 381.125,Z 587.898,A -85,B 0,C 180,E1 12453.521,E2 12453.521} C_VEL
LIN {X 0,Y 379.718,Z 584.063,A -85,B 0,C 180,E1 12455.194,E2 12455.194} C_VEL
LIN {X 0,Y 379.686,Z 582.416,A -85,B 0,C 180,E1 12457.276,E2 12457.276} C_VEL
LIN {X 0,Y 381.65,Z 587.263,A -85,B 0,C 180,E1 12459.674,E2 12459.674} C_VEL
LIN {X 0,Y 386.123,Z 598.366,A -85,B 0,C 180,E1 12462.13,E2 12462.13} C_VEL
LIN {X 0,Y 392.413,Z 619.195,A -85,B 0,C 180,E1 12464.863,E2 12464.863} C_VEL
LIN {X 0,Y 395.541,Z 633.732,A -85,B 0,C 180,E1 12466.326,E2 12466.326} C_VEL
LIN {X 0,Y 388.422,Z 675.822,A -85,B 0,C 180,E1 12468.779,E2 12468.779} C_VEL
LIN {X 0,Y 380.801,Z 715.747,A -85,B 0,C 180,E1 12472.136,E2 12472.136} C_VEL
LIN {X 0,Y 373.618,Z 750.775,A -85,B 0,C 180,E1 12476.221,E2 12476.221} C_VEL
LIN {X 0,Y 367.375,Z 781.304,A -85,B 0,C 180,E1 12481.035,E2 12481.035} C_VEL
LIN {X 0,Y 362.663,Z 805.632,A -85,B 0,C 180,E1 12486.181,E2 12486.181} C_VEL
LIN {X 0,Y 359.622,Z 825.368,A -85,B 0,C 180,E1 12491.889,E2 12491.889} C_VEL
LIN {X 0,Y 358.038,Z 839.483,A -85,B 0,C 180,E1 12497.792,E2 12497.792} C_VEL
LIN {X 0,Y 357.53,Z 848.083,A -85,B 0,C 180,E1 12503.774,E2 12503.774} C_VEL
LIN {X 0,Y 357.468,Z 849.861,A -85,B 0,C 180,E1 12506.174,E2 12506.174} C_VEL
LIN {X 0,Y 354.982,Z 850.689,A -85,B 0,C 180,E1 12508.243,E2 12508.243} C_VEL
LIN {X 0,Y 349.695,Z 850.283,A -85,B 0,C 180,E1 12511.733,E2 12511.733} C_VEL
LIN {X 0,Y 349.727,Z 846.819,A -85,B 0,C 180,E1 12517.461,E2 12517.461} C_VEL
LIN {X 0,Y 350.374,Z 838.558,A -85,B 0,C 180,E1 12523.23,E2 12523.23} C_VEL
LIN {X 0,Y 352.271,Z 824.092,A -85,B 0,C 180,E1 12529.422,E2 12529.422} C_VEL
LIN {X 0,Y 356.272,Z 803.612,A -85,B 0,C 180,E1 12535.441,E2 12535.441} C_VEL
LIN {X 0,Y 361.971,Z 778.679,A -85,B 0,C 180,E1 12540.741,E2 12540.741} C_VEL
LIN {X 0,Y 369.057,Z 748.957,A -85,B 0,C 180,E1 12545.413,E2 12545.413} C_VEL
LIN {X 0,Y 376.743,Z 715.548,A -85,B 0,C 180,E1 12549.268,E2 12549.268} C_VEL
LIN {X 0,Y 384.266,Z 678.053,A -85,B 0,C 180,E1 12552.368,E2 12552.368} C_VEL
LIN {X 0,Y 390.878,Z 636.641,A -85,B 0,C 180,E1 12554.642,E2 12554.642} C_VEL
LIN {X 0,Y 377.337,Z 604.715,A -85,B 0,C 180,E1 12557.876,E2 12557.876} C_VEL
LIN {X 0,Y 355.332,Z 564.778,A -85,B 0,C 180,E1 12562.429,E2 12562.429} C_VEL
LIN {X 0,Y 347.593,Z 550.248,A -85,B 0,C 180,E1 12564.203,E2 12564.203} C_VEL
LIN {X 0,Y 347.706,Z 549.53,A -85,B 0,C 180,E1 12571.387,E2 12571.387} C_VEL
LIN {X 0,Y 348.05,Z 549.53,A -85,B 0,C 180,E1 12579.64,E2 12579.64} C_VEL
LIN {X 0,Y 348.284,Z 549.53,A -85,B 0,C 180,E1 12584.886,E2 12584.886} C_VEL
LIN {X 0,Y 348.722,Z 549.53,A -85,B 0,C 180,E1 12592.521,E2 12592.521} C_VEL
LIN {X 0,Y 349.183,Z 549.53,A -85,B 0,C 180,E1 12600.005,E2 12600.005} C_VEL
LIN {X 0,Y 348.79,Z 549.53,A -85,B 0,C 180,E1 12607.488,E2 12607.488} C_VEL
LIN {X 0,Y 348.298,Z 549.53,A -85,B 0,C 180,E1 12615.124,E2 12615.124} C_VEL
LIN {X 0,Y 347.9,Z 549.53,A -85,B 0,C 180,E1 12623.064,E2 12623.064} C_VEL
LIN {X 0,Y 347.644,Z 549.53,A -85,B 0,C 180,E1 12629.422,E2 12629.422} C_VEL
LIN {X 0,Y 347.506,Z 549.53,A -85,B 0,C 180,E1 12634.505,E2 12634.505} C_VEL
LIN {X 0,Y 347.349,Z 549.53,A -85,B 0,C 180,E1 12642.184,E2 12642.184} C_VEL
LIN {X 0,Y 347.335,Z 549.53,A -85,B 0,C 180,E1 12649.168,E2 12649.168} C_VEL
LIN {X 0,Y 347.556,Z 549.53,A -85,B 0,C 180,E1 12655.87,E2 12655.87} C_VEL
LIN {X 0,Y 347.697,Z 549.53,A -85,B 0,C 180,E1 12661.381,E2 12661.381} C_VEL
LIN {X 0,Y 348.076,Z 549.53,A -85,B 0,C 180,E1 12669.637,E2 12669.637} C_VEL
LIN {X 0,Y 348.316,Z 549.53,A -85,B 0,C 180,E1 12674.883,E2 12674.883} C_VEL
LIN {X 0,Y 348.752,Z 549.53,A -85,B 0,C 180,E1 12682.518,E2 12682.518} C_VEL
LIN {X 0,Y 349.26,Z 549.53,A -85,B 0,C 180,E1 12690.001,E2 12690.001} C_VEL
LIN {X 0,Y 348.815,Z 549.53,A -85,B 0,C 180,E1 12697.483,E2 12697.483} C_VEL
LIN {X 0,Y 348.321,Z 549.53,A -85,B 0,C 180,E1 12705.119,E2 12705.119} C_VEL
LIN {X 0,Y 348.041,Z 549.885,A -85,B 0,C 180,E1 12712.809,E2 12712.809} C_VEL
LIN {X 0,Y 355.407,Z 565.268,A -85,B 0,C 180,E1 12714.803,E2 12714.803} C_VEL
LIN {X 0,Y 369.988,Z 597.398,A -85,B 0,C 180,E1 12719.076,E2 12719.076} C_VEL
LIN {X 0,Y 380.633,Z 628.98,A -85,B 0,C 180,E1 12723.227,E2 12723.227} C_VEL
LIN {X 0,Y 382.313,Z 638.488,A -85,B 0,C 180,E1 12724.416,E2 12724.416} C_VEL
LIN {X 0,Y 374.672,Z 673.772,A -85,B 0,C 180,E1 12728.02,E2 12728.02} C_VEL
LIN {X 0,Y 367.025,Z 704.823,A -85,B 0,C 180,E1 12732.422,E2 12732.422} C_VEL
LIN {X 0,Y 360.452,Z 730.086,A -85,B 0,C 180,E1 12737.279,E2 12737.279} C_VEL
LIN {X 0,Y 355.22,Z 751.295,A -85,B 0,C 180,E1 12742.881,E2 12742.881} C_VEL
LIN {X 0,Y 351.899,Z 767.328,A -85,B 0,C 180,E1 12748.91,E2 12748.91} C_VEL
LIN {X 0,Y 350.213,Z 778.177,A -85,B 0,C 180,E1 12755.217,E2 12755.217} C_VEL
LIN {X 0,Y 349.533,Z 782.689,A -85,B 0,C 180,E1 12759.72,E2 12759.72} C_VEL
LIN {X 0,Y 349.204,Z 784.785,A -85,B 0,C 180,E1 12764.916,E2 12764.916} C_VEL
LIN {X 0,Y 349.61,Z 783.431,A -85,B 0,C 180,E1 12770.019,E2 12770.019} C_VEL
LIN {X 0,Y 350.789,Z 777.401,A -85,B 0,C 180,E1 12776.283,E2 12776.283} C_VEL
LIN {X 0,Y 353.006,Z 766.357,A -85,B 0,C 180,E1 12782.453,E2 12782.453} C_VEL
LIN {X 0,Y 357.09,Z 749.694,A -85,B 0,C 180,E1 12788.529,E2 12788.529} C_VEL
LIN {X 0,Y 362.958,Z 728.828,A -85,B 0,C 180,E1 12793.873,E2 12793.873} C_VEL
LIN {X 0,Y 370.33,Z 702.49,A -85,B 0,C 180,E1 12798.776,E2 12798.776} C_VEL
LIN {X 0,Y 378.379,Z 671.707,A -85,B 0,C 180,E1 12802.959,E2 12802.959} C_VEL
LIN {X 0,Y 385.777,Z 638.133,A -85,B 0,C 180,E1 12806.303,E2 12806.303} C_VEL
LIN {X 0,Y 381.101,Z 607.713,A -85,B 0,C 180,E1 12810.88,E2 12810.88} C_VEL
LIN {X 0,Y 378.285,Z 595.907,A -85,B 0,C 180,E1 12813.516,E2 12813.516} C_VEL
LIN {X 0,Y 377.129,Z 591.309,A -85,B 0,C 180,E1 12815.472,E2 12815.472} C_VEL
LIN {X 0,Y 377.334,Z 589.747,A -85,B 0,C 180,E1 12816.997,E2 12816.997} C_VEL
LIN {X 0,Y 379.016,Z 595.004,A -85,B 0,C 180,E1 12819.563,E2 12819.563} C_VEL
LIN {X 0,Y 382.688,Z 605.942,A -85,B 0,C 180,E1 12821.914,E2 12821.914} C_VEL
LIN {X 0,Y 387.632,Z 625.782,A -85,B 0,C 180,E1 12824.526,E2 12824.526} C_VEL
LIN {X 0,Y 389.264,Z 637.695,A -85,B 0,C 180,E1 12825.701,E2 12825.701} C_VEL
LIN {X 0,Y 381.433,Z 679.926,A -85,B 0,C 180,E1 12828.334,E2 12828.334} C_VEL
LIN {X 0,Y 373.445,Z 718.829,A -85,B 0,C 180,E1 12831.808,E2 12831.808} C_VEL
LIN {X 0,Y 366.103,Z 752.406,A -85,B 0,C 180,E1 12835.898,E2 12835.898} C_VEL
LIN {X 0,Y 359.778,Z 781.806,A -85,B 0,C 180,E1 12840.71,E2 12840.71} C_VEL
LIN {X 0,Y 354.89,Z 805.748,A -85,B 0,C 180,E1 12845.95,E2 12845.95} C_VEL
LIN {X 0,Y 351.764,Z 825.203,A -85,B 0,C 180,E1 12851.768,E2 12851.768} C_VEL
LIN {X 0,Y 350.199,Z 838.621,A -85,B 0,C 180,E1 12857.515,E2 12857.515} C_VEL
LIN {X 0,Y 349.767,Z 846.102,A -85,B 0,C 180,E1 12862.537,E2 12862.537} C_VEL
LIN {X 0,Y 349.708,Z 849.949,A -85,B 0,C 180,E1 12867.518,E2 12867.518} C_VEL
LIN {X 0,Y 349.695,Z 850.283,A -85,B 0,C 180,E1 12871.733,E2 12871.733} C_VEL
LIN {X 0,Y 347.145,Z 849.386,A -85,B 0,C 180,E1 12873.845,E2 12873.845} C_VEL
LIN {X 0,Y 341.86,Z 846.673,A -85,B 0,C 180,E1 12877.012,E2 12877.012} C_VEL
LIN {X 0,Y 341.809,Z 846.299,A -85,B 0,C 180,E1 12877.378,E2 12877.378} C_VEL
LIN {X 0,Y 342.548,Z 837.769,A -85,B 0,C 180,E1 12883.521,E2 12883.521} C_VEL
LIN {X 0,Y 344.611,Z 822.93,A -85,B 0,C 180,E1 12889.959,E2 12889.959} C_VEL
LIN {X 0,Y 348.574,Z 803.623,A -85,B 0,C 180,E1 12895.743,E2 12895.743} C_VEL
LIN {X 0,Y 354.627,Z 778.225,A -85,B 0,C 180,E1 12901.277,E2 12901.277} C_VEL
LIN {X 0,Y 362.045,Z 748.605,A -85,B 0,C 180,E1 12906.016,E2 12906.016} C_VEL
LIN {X 0,Y 370.043,Z 715.103,A -85,B 0,C 180,E1 12909.93,E2 12909.93} C_VEL
LIN {X 0,Y 377.827,Z 677.587,A -85,B 0,C 180,E1 12913.073,E2 12913.073} C_VEL
LIN {X 0,Y 384.105,Z 638.088,A -85,B 0,C 180,E1 12915.332,E2 12915.332} C_VEL
LIN {X 0,Y 368.895,Z 603.213,A -85,B 0,C 180,E1 12919.057,E2 12919.057} C_VEL
LIN {X 0,Y 344.681,Z 559.984,A -85,B 0,C 180,E1 12924.318,E2 12924.318} C_VEL
LIN {X 0,Y 339.694,Z 550.109,A -85,B 0,C 180,E1 12925.547,E2 12925.547} C_VEL
LIN {X 0,Y 339.758,Z 549.53,A -85,B 0,C 180,E1 12933.03,E2 12933.03} C_VEL
LIN {X 0,Y 340.074,Z 549.53,A -85,B 0,C 180,E1 12939.218,E2 12939.218} C_VEL
LIN {X 0,Y 340.51,Z 549.53,A -85,B 0,C 180,E1 12947.16,E2 12947.16} C_VEL
LIN {X 0,Y 340.989,Z 549.53,A -85,B 0,C 180,E1 12954.911,E2 12954.911} C_VEL
LIN {X 0,Y 341.297,Z 549.53,A -85,B 0,C 180,E1 12960.005,E2 12960.005} C_VEL
LIN {X 0,Y 340.848,Z 549.53,A -85,B 0,C 180,E1 12967.663,E2 12967.663} C_VEL
LIN {X 0,Y 340.366,Z 549.53,A -85,B 0,C 180,E1 12975.485,E2 12975.485} C_VEL
LIN {X 0,Y 339.946,Z 549.53,A -85,B 0,C 180,E1 12983.636,E2 12983.636} C_VEL
LIN {X 0,Y 339.747,Z 549.53,A -85,B 0,C 180,E1 12989.36,E2 12989.36} C_VEL
LIN {X 0,Y 339.428,Z 549.53,A -85,B 0,C 180,E1 12996.593,E2 12996.593} C_VEL
LIN {X 0,Y 339.441,Z 549.53,A -85,B 0,C 180,E1 13002.001,E2 13002.001} C_VEL
LIN {X 0,Y 339.418,Z 549.53,A -85,B 0,C 180,E1 13009.324,E2 13009.324} C_VEL
LIN {X 0,Y 339.651,Z 549.53,A -85,B 0,C 180,E1 13017.662,E2 13017.662} C_VEL
LIN {X 0,Y 339.81,Z 549.53,A -85,B 0,C 180,E1 13023.542,E2 13023.542} C_VEL
LIN {X 0,Y 340.26,Z 549.53,A -85,B 0,C 180,E1 13031.853,E2 13031.853} C_VEL
LIN {X 0,Y 340.652,Z 549.53,A -85,B 0,C 180,E1 13039.76,E2 13039.76} C_VEL
LIN {X 0,Y 341.252,Z 549.53,A -85,B 0,C 180,E1 13047.458,E2 13047.458} C_VEL
LIN {X 0,Y 341.268,Z 549.53,A -85,B 0,C 180,E1 13052.544,E2 13052.544} C_VEL
LIN {X 0,Y 340.635,Z 549.53,A -85,B 0,C 180,E1 13060.242,E2 13060.242} C_VEL
LIN {X 0,Y 340.274,Z 549.53,A -85,B 0,C 180,E1 13068.149,E2 13068.149} C_VEL
LIN {X 0,Y 340.102,Z 549.53,A -85,B 0,C 180,E1 13071.462,E2 13071.462} C_VEL
LIN {X 0,Y 344.818,Z 559.895,A -85,B 0,C 180,E1 13072.816,E2 13072.816} C_VEL
LIN {X 0,Y 360.074,Z 591.968,A -85,B 0,C 180,E1 13077.291,E2 13077.291} C_VEL
LIN {X 0,Y 371.295,Z 622.513,A -85,B 0,C 180,E1 13081.464,E2 13081.464} C_VEL
LIN {X 0,Y 375.542,Z 640.454,A -85,B 0,C 180,E1 13083.856,E2 13083.856} C_VEL
LIN {X 0,Y 367.559,Z 675.826,A -85,B 0,C 180,E1 13087.566,E2 13087.566} C_VEL
LIN {X 0,Y 359.746,Z 706.424,A -85,B 0,C 180,E1 13092.013,E2 13092.013} C_VEL
LIN {X 0,Y 353.154,Z 730.752,A -85,B 0,C 180,E1 13096.79,E2 13096.79} C_VEL
LIN {X 0,Y 347.726,Z 751.804,A -85,B 0,C 180,E1 13102.435,E2 13102.435} C_VEL
LIN {X 0,Y 344.369,Z 767.022,A -85,B 0,C 180,E1 13108.152,E2 13108.152} C_VEL
LIN {X 0,Y 342.669,Z 777.179,A -85,B 0,C 180,E1 13113.773,E2 13113.773} C_VEL
LIN {X 0,Y 341.725,Z 783.111,A -85,B 0,C 180,E1 13119.235,E2 13119.235} C_VEL
LIN {X 0,Y 341.311,Z 785.466,A -85,B 0,C 180,E1 13124.559,E2 13124.559} C_VEL
LIN {X 0,Y 341.733,Z 784.442,A -85,B 0,C 180,E1 13129.787,E2 13129.787} C_VEL
LIN {X 0,Y 342.954,Z 778.718,A -85,B 0,C 180,E1 13136.198,E2 13136.198} C_VEL
LIN {X 0,Y 345.26,Z 768.022,A -85,B 0,C 180,E1 13142.508,E2 13142.508} C_VEL
LIN {X 0,Y 349.523,Z 751.733,A -85,B 0,C 180,E1 13148.715,E2 13148.715} C_VEL
LIN {X 0,Y 355.607,Z 731.314,A -85,B 0,C 180,E1 13154.165,E2 13154.165} C_VEL
LIN {X 0,Y 363.288,Z 705.589,A -85,B 0,C 180,E1 13159.154,E2 13159.154} C_VEL
LIN {X 0,Y 371.647,Z 675.621,A -85,B 0,C 180,E1 13163.399,E2 13163.399} C_VEL
LIN {X 0,Y 379.844,Z 640.825,A -85,B 0,C 180,E1 13167.052,E2 13167.052} C_VEL
LIN {X 0,Y 376.695,Z 612.887,A -85,B 0,C 180,E1 13171.494,E2 13171.494} C_VEL
LIN {X 0,Y 374.788,Z 601.068,A -85,B 0,C 180,E1 13174.435,E2 13174.435} C_VEL
LIN {X 0,Y 374.523,Z 598.161,A -85,B 0,C 180,E1 13176.046,E2 13176.046} C_VEL
LIN {X 0,Y 374.859,Z 597.82,A -85,B 0,C 180,E1 13177.283,E2 13177.283} C_VEL
LIN {X 0,Y 376.423,Z 603.306,A -85,B 0,C 180,E1 13179.623,E2 13179.623} C_VEL
LIN {X 0,Y 379.847,Z 617.26,A -85,B 0,C 180,E1 13182.268,E2 13182.268} C_VEL
LIN {X 0,Y 383.699,Z 638.498,A -85,B 0,C 180,E1 13184.884,E2 13184.884} C_VEL
LIN {X 0,Y 375.08,Z 681.11,A -85,B 0,C 180,E1 13187.65,E2 13187.65} C_VEL
LIN {X 0,Y 366.399,Z 720.626,A -85,B 0,C 180,E1 13191.316,E2 13191.316} C_VEL
LIN {X 0,Y 358.439,Z 754.915,A -85,B 0,C 180,E1 13195.679,E2 13195.679} C_VEL
LIN {X 0,Y 351.399,Z 785.635,A -85,B 0,C 180,E1 13201.004,E2 13201.004} C_VEL
LIN {X 0,Y 346.382,Z 810.111,A -85,B 0,C 180,E1 13206.833,E2 13206.833} C_VEL
LIN {X 0,Y 343.46,Z 827.896,A -85,B 0,C 180,E1 13212.688,E2 13212.688} C_VEL
LIN {X 0,Y 342.193,Z 840.017,A -85,B 0,C 180,E1 13218.514,E2 13218.514} C_VEL
LIN {X 0,Y 341.797,Z 846.635,A -85,B 0,C 180,E1 13223.641,E2 13223.641} C_VEL
LIN {X 0,Y 341.967,Z 849.789,A -85,B 0,C 180,E1 13229.999,E2 13229.999} C_VEL
LIN {X 0,Y 341.735,Z 847.278,A -85,B 0,C 180,E1 13236.358,E2 13236.358} C_VEL
LIN {X 0,Y 341.809,Z 846.299,A -85,B 0,C 180,E1 13237.378,E2 13237.378} C_VEL
LIN {X 0,Y 339.492,Z 843.815,A -85,B 0,C 180,E1 13239.506,E2 13239.506} C_VEL
LIN {X 0,Y 334.556,Z 838.935,A -85,B 0,C 180,E1 13242.683,E2 13242.683} C_VEL
LIN {X 0,Y 334.542,Z 838.358,A -85,B 0,C 180,E1 13243.049,E2 13243.049} C_VEL
LIN {X 0,Y 336.438,Z 824.909,A -85,B 0,C 180,E1 13249.352,E2 13249.352} C_VEL
LIN {X 0,Y 340.554,Z 805.084,A -85,B 0,C 180,E1 13255.687,E2 13255.687} C_VEL
LIN {X 0,Y 346.592,Z 780.815,A -85,B 0,C 180,E1 13261.247,E2 13261.247} C_VEL
LIN {X 0,Y 354.412,Z 750.595,A -85,B 0,C 180,E1 13266.296,E2 13266.296} C_VEL
LIN {X 0,Y 362.629,Z 717.507,A -85,B 0,C 180,E1 13270.327,E2 13270.327} C_VEL
LIN {X 0,Y 370.496,Z 681.677,A -85,B 0,C 180,E1 13273.471,E2 13273.471} C_VEL
LIN {X 0,Y 377.594,Z 642.231,A -85,B 0,C 180,E1 13275.831,E2 13275.831} C_VEL
LIN {X 0,Y 366.085,Z 613.314,A -85,B 0,C 180,E1 13278.97,E2 13278.97} C_VEL
LIN {X 0,Y 345.724,Z 575.214,A -85,B 0,C 180,E1 13283.569,E2 13283.569} C_VEL
LIN {X 0,Y 331.847,Z 550.884,A -85,B 0,C 180,E1 13286.919,E2 13286.919} C_VEL
LIN {X 0,Y 331.728,Z 549.53,A -85,B 0,C 180,E1 13287.108,E2 13287.108} C_VEL
LIN {X 0,Y 331.869,Z 549.53,A -85,B 0,C 180,E1 13292.863,E2 13292.863} C_VEL
LIN {X 0,Y 332.25,Z 549.53,A -85,B 0,C 180,E1 13301.404,E2 13301.404} C_VEL
LIN {X 0,Y 332.694,Z 549.53,A -85,B 0,C 180,E1 13309.517,E2 13309.517} C_VEL
LIN {X 0,Y 333.264,Z 549.53,A -85,B 0,C 180,E1 13317.402,E2 13317.402} C_VEL
LIN {X 0,Y 333.347,Z 549.53,A -85,B 0,C 180,E1 13322.609,E2 13322.609} C_VEL
LIN {X 0,Y 332.676,Z 549.53,A -85,B 0,C 180,E1 13330.494,E2 13330.494} C_VEL
LIN {X 0,Y 332.274,Z 549.53,A -85,B 0,C 180,E1 13338.606,E2 13338.606} C_VEL
LIN {X 0,Y 331.876,Z 549.53,A -85,B 0,C 180,E1 13347.148,E2 13347.148} C_VEL
LIN {X 0,Y 331.537,Z 549.53,A -85,B 0,C 180,E1 13354.714,E2 13354.714} C_VEL
LIN {X 0,Y 331.519,Z 549.53,A -85,B 0,C 180,E1 13359.752,E2 13359.752} C_VEL
LIN {X 0,Y 331.466,Z 549.53,A -85,B 0,C 180,E1 13366.964,E2 13366.964} C_VEL
LIN {X 0,Y 331.551,Z 549.53,A -85,B 0,C 180,E1 13373.584,E2 13373.584} C_VEL
LIN {X 0,Y 331.775,Z 549.53,A -85,B 0,C 180,E1 13380.128,E2 13380.128} C_VEL
LIN {X 0,Y 332.104,Z 549.53,A -85,B 0,C 180,E1 13388.611,E2 13388.611} C_VEL
LIN {X 0,Y 332.42,Z 549.53,A -85,B 0,C 180,E1 13394.142,E2 13394.142} C_VEL
LIN {X 0,Y 332.894,Z 549.53,A -85,B 0,C 180,E1 13402.159,E2 13402.159} C_VEL
LIN {X 0,Y 333.47,Z 549.53,A -85,B 0,C 180,E1 13410.001,E2 13410.001} C_VEL
LIN {X 0,Y 332.941,Z 549.53,A -85,B 0,C 180,E1 13417.842,E2 13417.842} C_VEL
LIN {X 0,Y 332.428,Z 549.53,A -85,B 0,C 180,E1 13425.86,E2 13425.86} C_VEL
LIN {X 0,Y 332.226,Z 549.53,A -85,B 0,C 180,E1 13430.081,E2 13430.081} C_VEL
LIN {X 0,Y 334.659,Z 555.175,A -85,B 0,C 180,E1 13430.85,E2 13430.85} C_VEL
LIN {X 0,Y 350.548,Z 587.705,A -85,B 0,C 180,E1 13435.59,E2 13435.59} C_VEL
LIN {X 0,Y 362.782,Z 619.31,A -85,B 0,C 180,E1 13440.055,E2 13440.055} C_VEL
LIN {X 0,Y 368.809,Z 642.287,A -85,B 0,C 180,E1 13443.268,E2 13443.268} C_VEL
LIN {X 0,Y 360.53,Z 677.55,A -85,B 0,C 180,E1 13447.062,E2 13447.062} C_VEL
LIN {X 0,Y 352.669,Z 707.233,A -85,B 0,C 180,E1 13451.46,E2 13451.46} C_VEL
LIN {X 0,Y 345.715,Z 731.965,A -85,B 0,C 180,E1 13456.41,E2 13456.41} C_VEL
LIN {X 0,Y 340.203,Z 752.484,A -85,B 0,C 180,E1 13462.033,E2 13462.033} C_VEL
LIN {X 0,Y 336.53,Z 768.326,A -85,B 0,C 180,E1 13468.156,E2 13468.156} C_VEL
LIN {X 0,Y 334.746,Z 778.544,A -85,B 0,C 180,E1 13474.05,E2 13474.05} C_VEL
LIN {X 0,Y 333.935,Z 783.53,A -85,B 0,C 180,E1 13478.727,E2 13478.727} C_VEL
LIN {X 0,Y 333.435,Z 786.146,A -85,B 0,C 180,E1 13484.185,E2 13484.185} C_VEL
LIN {X 0,Y 333.825,Z 785.453,A -85,B 0,C 180,E1 13489.542,E2 13489.542} C_VEL
LIN {X 0,Y 335.122,Z 780.057,A -85,B 0,C 180,E1 13496.109,E2 13496.109} C_VEL
LIN {X 0,Y 337.498,Z 769.709,A -85,B 0,C 180,E1 13502.566,E2 13502.566} C_VEL
LIN {X 0,Y 341.953,Z 753.83,A -85,B 0,C 180,E1 13508.909,E2 13508.909} C_VEL
LIN {X 0,Y 348.69,Z 732.574,A -85,B 0,C 180,E1 13514.774,E2 13514.774} C_VEL
LIN {X 0,Y 356.794,Z 707.059,A -85,B 0,C 180,E1 13519.839,E2 13519.839} C_VEL
LIN {X 0,Y 365.7,Z 677.113,A -85,B 0,C 180,E1 13524.18,E2 13524.18} C_VEL
LIN {X 0,Y 374.175,Z 644.556,A -85,B 0,C 180,E1 13527.676,E2 13527.676} C_VEL
LIN {X 0,Y 372.379,Z 617.822,A -85,B 0,C 180,E1 13532.185,E2 13532.185} C_VEL
LIN {X 0,Y 371.73,Z 608.092,A -85,B 0,C 180,E1 13534.759,E2 13534.759} C_VEL
LIN {X 0,Y 371.795,Z 606.388,A -85,B 0,C 180,E1 13535.464,E2 13535.464} C_VEL
LIN {X 0,Y 372.21,Z 605.896,A -85,B 0,C 180,E1 13537.594,E2 13537.594} C_VEL
LIN {X 0,Y 373.376,Z 611.468,A -85,B 0,C 180,E1 13539.603,E2 13539.603} C_VEL
LIN {X 0,Y 376.267,Z 627.903,A -85,B 0,C 180,E1 13542.482,E2 13542.482} C_VEL
LIN {X 0,Y 377.614,Z 642.756,A -85,B 0,C 180,E1 13544.216,E2 13544.216} C_VEL
LIN {X 0,Y 368.032,Z 686.369,A -85,B 0,C 180,E1 13547.25,E2 13547.25} C_VEL
LIN {X 0,Y 358.607,Z 725.842,A -85,B 0,C 180,E1 13551.181,E2 13551.181} C_VEL
LIN {X 0,Y 350.241,Z 759.604,A -85,B 0,C 180,E1 13555.806,E2 13555.806} C_VEL
LIN {X 0,Y 343.417,Z 787.673,A -85,B 0,C 180,E1 13560.988,E2 13560.988} C_VEL
LIN {X 0,Y 338.609,Z 810.262,A -85,B 0,C 180,E1 13566.618,E2 13566.618} C_VEL
LIN {X 0,Y 335.72,Z 826.997,A -85,B 0,C 180,E1 13572.276,E2 13572.276} C_VEL
LIN {X 0,Y 334.355,Z 839.185,A -85,B 0,C 180,E1 13578.241,E2 13578.241} C_VEL
LIN {X 0,Y 333.939,Z 845.851,A -85,B 0,C 180,E1 13583.49,E2 13583.49} C_VEL
LIN {X 0,Y 333.976,Z 848.436,A -85,B 0,C 180,E1 13587.401,E2 13587.401} C_VEL
LIN {X 0,Y 334.002,Z 848.664,A -85,B 0,C 180,E1 13592.597,E2 13592.597} C_VEL
LIN {X 0,Y 334.066,Z 843.908,A -85,B 0,C 180,E1 13599.126,E2 13599.126} C_VEL
LIN {X 0,Y 334.542,Z 838.358,A -85,B 0,C 180,E1 13603.049,E2 13603.049} C_VEL
LIN {X 0,Y 332.511,Z 834.535,A -85,B 0,C 180,E1 13605.18,E2 13605.18} C_VEL
LIN {X 0,Y 328.174,Z 827.593,A -85,B 0,C 180,E1 13608.327,E2 13608.327} C_VEL
LIN {X 0,Y 328.234,Z 826.731,A -85,B 0,C 180,E1 13608.683,E2 13608.683} C_VEL
LIN {X 0,Y 331.95,Z 808.676,A -85,B 0,C 180,E1 13614.954,E2 13614.954} C_VEL
LIN {X 0,Y 337.693,Z 786.092,A -85,B 0,C 180,E1 13620.594,E2 13620.594} C_VEL
LIN {X 0,Y 345.065,Z 758.663,A -85,B 0,C 180,E1 13625.65,E2 13625.65} C_VEL
LIN {X 0,Y 353.529,Z 726.739,A -85,B 0,C 180,E1 13629.97,E2 13629.97} C_VEL
LIN {X 0,Y 362.12,Z 690.514,A -85,B 0,C 180,E1 13633.495,E2 13633.495} C_VEL
LIN {X 0,Y 369.923,Z 651.224,A -85,B 0,C 180,E1 13636.116,E2 13636.116} C_VEL
LIN {X 0,Y 370.521,Z 642.196,A -85,B 0,C 180,E1 13636.674,E2 13636.674} C_VEL
LIN {X 0,Y 355.601,Z 607.428,A -85,B 0,C 180,E1 13640.711,E2 13640.711} C_VEL
LIN {X 0,Y 332.444,Z 565.752,A -85,B 0,C 180,E1 13646.198,E2 13646.198} C_VEL
LIN {X 0,Y 324.044,Z 551.312,A -85,B 0,C 180,E1 13648.359,E2 13648.359} C_VEL
LIN {X 0,Y 323.86,Z 549.53,A -85,B 0,C 180,E1 13648.649,E2 13648.649} C_VEL
LIN {X 0,Y 323.955,Z 549.53,A -85,B 0,C 180,E1 13655.132,E2 13655.132} C_VEL
LIN {X 0,Y 324.262,Z 549.53,A -85,B 0,C 180,E1 13660.929,E2 13660.929} C_VEL
LIN {X 0,Y 324.747,Z 549.53,A -85,B 0,C 180,E1 13669.258,E2 13669.258} C_VEL
LIN {X 0,Y 325.347,Z 549.53,A -85,B 0,C 180,E1 13677.338,E2 13677.338} C_VEL
LIN {X 0,Y 325.427,Z 549.53,A -85,B 0,C 180,E1 13682.672,E2 13682.672} C_VEL
LIN {X 0,Y 324.726,Z 549.53,A -85,B 0,C 180,E1 13690.754,E2 13690.754} C_VEL
LIN {X 0,Y 324.472,Z 549.53,A -85,B 0,C 180,E1 13696.264,E2 13696.264} C_VEL
LIN {X 0,Y 324.144,Z 549.53,A -85,B 0,C 180,E1 13701.948,E2 13701.948} C_VEL
LIN {X 0,Y 323.886,Z 549.53,A -85,B 0,C 180,E1 13707.876,E2 13707.876} C_VEL
LIN {X 0,Y 323.628,Z 549.53,A -85,B 0,C 180,E1 13714.159,E2 13714.159} C_VEL
LIN {X 0,Y 323.463,Z 549.53,A -85,B 0,C 180,E1 13721.504,E2 13721.504} C_VEL
LIN {X 0,Y 323.461,Z 549.53,A -85,B 0,C 180,E1 13729.058,E2 13729.058} C_VEL
LIN {X 0,Y 323.642,Z 549.53,A -85,B 0,C 180,E1 13735.85,E2 13735.85} C_VEL
LIN {X 0,Y 323.935,Z 549.53,A -85,B 0,C 180,E1 13742.639,E2 13742.639} C_VEL
LIN {X 0,Y 324.295,Z 549.53,A -85,B 0,C 180,E1 13750.926,E2 13750.926} C_VEL
LIN {X 0,Y 324.774,Z 549.53,A -85,B 0,C 180,E1 13759.254,E2 13759.254} C_VEL
LIN {X 0,Y 325.449,Z 549.53,A -85,B 0,C 180,E1 13767.335,E2 13767.335} C_VEL
LIN {X 0,Y 325.451,Z 549.53,A -85,B 0,C 180,E1 13772.668,E2 13772.668} C_VEL
LIN {X 0,Y 324.748,Z 549.53,A -85,B 0,C 180,E1 13780.749,E2 13780.749} C_VEL
LIN {X 0,Y 324.399,Z 549.644,A -85,B 0,C 180,E1 13788.689,E2 13788.689} C_VEL
LIN {X 0,Y 326.762,Z 555.228,A -85,B 0,C 180,E1 13789.454,E2 13789.454} C_VEL
LIN {X 0,Y 343.025,Z 587.917,A -85,B 0,C 180,E1 13794.445,E2 13794.445} C_VEL
LIN {X 0,Y 355.786,Z 621.083,A -85,B 0,C 180,E1 13799.302,E2 13799.302} C_VEL
LIN {X 0,Y 361.987,Z 643.952,A -85,B 0,C 180,E1 13802.634,E2 13802.634} C_VEL
LIN {X 0,Y 353.648,Z 678.818,A -85,B 0,C 180,E1 13806.479,E2 13806.479} C_VEL
LIN {X 0,Y 345.421,Z 708.68,A -85,B 0,C 180,E1 13811.003,E2 13811.003} C_VEL
LIN {X 0,Y 338.125,Z 733.602,A -85,B 0,C 180,E1 13816.131,E2 13816.131} C_VEL
LIN {X 0,Y 332.333,Z 754.421,A -85,B 0,C 180,E1 13822.039,E2 13822.039} C_VEL
LIN {X 0,Y 328.744,Z 769.353,A -85,B 0,C 180,E1 13828.024,E2 13828.024} C_VEL
LIN {X 0,Y 326.866,Z 779.629,A -85,B 0,C 180,E1 13834.185,E2 13834.185} C_VEL
LIN {X 0,Y 326.156,Z 783.92,A -85,B 0,C 180,E1 13838.194,E2 13838.194} C_VEL
LIN {X 0,Y 325.571,Z 786.809,A -85,B 0,C 180,E1 13843.792,E2 13843.792} C_VEL
LIN {X 0,Y 325.917,Z 786.388,A -85,B 0,C 180,E1 13849.286,E2 13849.286} C_VEL
LIN {X 0,Y 327.267,Z 781.315,A -85,B 0,C 180,E1 13856.015,E2 13856.015} C_VEL
LIN {X 0,Y 330.112,Z 770.047,A -85,B 0,C 180,E1 13863.281,E2 13863.281} C_VEL
LIN {X 0,Y 334.956,Z 754.007,A -85,B 0,C 180,E1 13869.753,E2 13869.753} C_VEL
LIN {X 0,Y 342.237,Z 732.613,A -85,B 0,C 180,E1 13875.716,E2 13875.716} C_VEL
LIN {X 0,Y 350.962,Z 706.952,A -85,B 0,C 180,E1 13880.843,E2 13880.843} C_VEL
LIN {X 0,Y 360.839,Z 675.921,A -85,B 0,C 180,E1 13885.35,E2 13885.35} C_VEL
LIN {X 0,Y 368.628,Z 647.284,A -85,B 0,C 180,E1 13888.514,E2 13888.514} C_VEL
LIN {X 0,Y 368.355,Z 623.7,A -85,B 0,C 180,E1 13892.72,E2 13892.72} C_VEL
LIN {X 0,Y 368.57,Z 615.025,A -85,B 0,C 180,E1 13895.1,E2 13895.1} C_VEL
LIN {X 0,Y 368.764,Z 613.588,A -85,B 0,C 180,E1 13895.8,E2 13895.8} C_VEL
LIN {X 0,Y 369.509,Z 614.088,A -85,B 0,C 180,E1 13897.917,E2 13897.917} C_VEL
LIN {X 0,Y 370.407,Z 622.81,A -85,B 0,C 180,E1 13900.196,E2 13900.196} C_VEL
LIN {X 0,Y 372.424,Z 642.396,A -85,B 0,C 180,E1 13903.15,E2 13903.15} C_VEL
LIN {X 0,Y 361.41,Z 689.729,A -85,B 0,C 180,E1 13906.684,E2 13906.684} C_VEL
LIN {X 0,Y 351.471,Z 728.326,A -85,B 0,C 180,E1 13910.726,E2 13910.726} C_VEL
LIN {X 0,Y 342.393,Z 762.696,A -85,B 0,C 180,E1 13915.679,E2 13915.679} C_VEL
LIN {X 0,Y 335.115,Z 791.471,A -85,B 0,C 180,E1 13921.358,E2 13921.358} C_VEL
LIN {X 0,Y 330.184,Z 813.518,A -85,B 0,C 180,E1 13927.31,E2 13927.31} C_VEL
LIN {X 0,Y 327.354,Z 830.822,A -85,B 0,C 180,E1 13933.887,E2 13933.887} C_VEL
LIN {X 0,Y 326.24,Z 842.235,A -85,B 0,C 180,E1 13940.651,E2 13940.651} C_VEL
LIN {X 0,Y 326.124,Z 847.683,A -85,B 0,C 180,E1 13947.338,E2 13947.338} C_VEL
LIN {X 0,Y 326.146,Z 847.899,A -85,B 0,C 180,E1 13952.66,E2 13952.66} C_VEL
LIN {X 0,Y 326.094,Z 844.489,A -85,B 0,C 180,E1 13958.006,E2 13958.006} C_VEL
LIN {X 0,Y 327.006,Z 835.028,A -85,B 0,C 180,E1 13964.752,E2 13964.752} C_VEL
LIN {X 0,Y 328.234,Z 826.731,A -85,B 0,C 180,E1 13968.683,E2 13968.683} C_VEL
LIN {X 0,Y 326.749,Z 821.571,A -85,B 0,C 180,E1 13970.773,E2 13970.773} C_VEL
LIN {X 0,Y 323.299,Z 812.986,A -85,B 0,C 180,E1 13973.876,E2 13973.876} C_VEL
LIN {X 0,Y 323.438,Z 811.95,A -85,B 0,C 180,E1 13974.22,E2 13974.22} C_VEL
LIN {X 0,Y 329.734,Z 787.788,A -85,B 0,C 180,E1 13980.671,E2 13980.671} C_VEL
LIN {X 0,Y 337.722,Z 759.262,A -85,B 0,C 180,E1 13986.122,E2 13986.122} C_VEL
LIN {X 0,Y 346.378,Z 727.843,A -85,B 0,C 180,E1 13990.486,E2 13990.486} C_VEL
LIN {X 0,Y 355.163,Z 692.258,A -85,B 0,C 180,E1 13994.058,E2 13994.058} C_VEL
LIN {X 0,Y 362.985,Z 654.877,A -85,B 0,C 180,E1 13996.66,E2 13996.66} C_VEL
LIN {X 0,Y 364.171,Z 645.438,A -85,B 0,C 180,E1 13997.229,E2 13997.229} C_VEL
LIN {X 0,Y 349.328,Z 610.374,A -85,B 0,C 180,E1 14001.488,E2 14001.488} C_VEL
LIN {X 0,Y 327.738,Z 571.065,A -85,B 0,C 180,E1 14006.811,E2 14006.811} C_VEL
LIN {X 0,Y 316.036,Z 551.117,A -85,B 0,C 180,E1 14009.958,E2 14009.958} C_VEL
LIN {X 0,Y 315.846,Z 549.53,A -85,B 0,C 180,E1 14010.143,E2 14010.143} C_VEL
LIN {X 0,Y 316.091,Z 549.53,A -85,B 0,C 180,E1 14017.475,E2 14017.475} C_VEL
LIN {X 0,Y 316.47,Z 549.53,A -85,B 0,C 180,E1 14023.325,E2 14023.325} C_VEL
LIN {X 0,Y 316.984,Z 549.53,A -85,B 0,C 180,E1 14031.768,E2 14031.768} C_VEL
LIN {X 0,Y 317.611,Z 549.53,A -85,B 0,C 180,E1 14040.006,E2 14040.006} C_VEL
LIN {X 0,Y 317.232,Z 549.53,A -85,B 0,C 180,E1 14045.483,E2 14045.483} C_VEL
LIN {X 0,Y 316.629,Z 549.53,A -85,B 0,C 180,E1 14053.838,E2 14053.838} C_VEL
LIN {X 0,Y 316.342,Z 549.53,A -85,B 0,C 180,E1 14059.58,E2 14059.58} C_VEL
LIN {X 0,Y 316.034,Z 549.53,A -85,B 0,C 180,E1 14065.548,E2 14065.548} C_VEL
LIN {X 0,Y 315.747,Z 549.53,A -85,B 0,C 180,E1 14071.841,E2 14071.841} C_VEL
LIN {X 0,Y 315.498,Z 549.53,A -85,B 0,C 180,E1 14079.842,E2 14079.842} C_VEL
LIN {X 0,Y 315.472,Z 549.53,A -85,B 0,C 180,E1 14087.787,E2 14087.787} C_VEL
LIN {X 0,Y 315.616,Z 549.53,A -85,B 0,C 180,E1 14094.856,E2 14094.856} C_VEL
LIN {X 0,Y 315.86,Z 549.53,A -85,B 0,C 180,E1 14101.359,E2 14101.359} C_VEL
LIN {X 0,Y 316.111,Z 549.53,A -85,B 0,C 180,E1 14107.471,E2 14107.471} C_VEL
LIN {X 0,Y 316.506,Z 549.53,A -85,B 0,C 180,E1 14113.322,E2 14113.322} C_VEL
LIN {X 0,Y 317.013,Z 549.53,A -85,B 0,C 180,E1 14121.763,E2 14121.763} C_VEL
LIN {X 0,Y 317.704,Z 549.53,A -85,B 0,C 180,E1 14130.001,E2 14130.001} C_VEL
LIN {X 0,Y 317.047,Z 549.53,A -85,B 0,C 180,E1 14138.238,E2 14138.238} C_VEL
LIN {X 0,Y 316.525,Z 549.53,A -85,B 0,C 180,E1 14146.912,E2 14146.912} C_VEL
LIN {X 0,Y 316.917,Z 552.049,A -85,B 0,C 180,E1 14147.384,E2 14147.384} C_VEL
LIN {X 0,Y 333.131,Z 583.206,A -85,B 0,C 180,E1 14152.478,E2 14152.478} C_VEL
LIN {X 0,Y 345.426,Z 613.018,A -85,B 0,C 180,E1 14157.05,E2 14157.05} C_VEL
LIN {X 0,Y 354.342,Z 642.47,A -85,B 0,C 180,E1 14161.491,E2 14161.491} C_VEL
LIN {X 0,Y 354.572,Z 649.402,A -85,B 0,C 180,E1 14162.396,E2 14162.396} C_VEL
LIN {X 0,Y 345.947,Z 683.018,A -85,B 0,C 180,E1 14166.271,E2 14166.271} C_VEL
LIN {X 0,Y 337.308,Z 713.093,A -85,B 0,C 180,E1 14171.061,E2 14171.061} C_VEL
LIN {X 0,Y 329.489,Z 738.88,A -85,B 0,C 180,E1 14176.759,E2 14176.759} C_VEL
LIN {X 0,Y 323.692,Z 759.343,A -85,B 0,C 180,E1 14183.144,E2 14183.144} C_VEL
LIN {X 0,Y 320.291,Z 773.771,A -85,B 0,C 180,E1 14189.692,E2 14189.692} C_VEL
LIN {X 0,Y 318.586,Z 782.827,A -85,B 0,C 180,E1 14196.169,E2 14196.169} C_VEL
LIN {X 0,Y 317.715,Z 787.176,A -85,B 0,C 180,E1 14202.386,E2 14202.386} C_VEL
LIN {X 0,Y 318.009,Z 787.308,A -85,B 0,C 180,E1 14209.016,E2 14209.016} C_VEL
LIN {X 0,Y 319.191,Z 783.546,A -85,B 0,C 180,E1 14214.966,E2 14214.966} C_VEL
LIN {X 0,Y 321.571,Z 774.181,A -85,B 0,C 180,E1 14222.018,E2 14222.018} C_VEL
LIN {X 0,Y 326.203,Z 759.743,A -85,B 0,C 180,E1 14228.67,E2 14228.67} C_VEL
LIN {X 0,Y 333.23,Z 740.25,A -85,B 0,C 180,E1 14234.802,E2 14234.802} C_VEL
LIN {X 0,Y 342.351,Z 715.346,A -85,B 0,C 180,E1 14240.376,E2 14240.376} C_VEL
LIN {X 0,Y 353.188,Z 684.015,A -85,B 0,C 180,E1 14245.378,E2 14245.378} C_VEL
LIN {X 0,Y 363.328,Z 651.513,A -85,B 0,C 180,E1 14249.148,E2 14249.148} C_VEL
LIN {X 0,Y 364.546,Z 628.474,A -85,B 0,C 180,E1 14253.54,E2 14253.54} C_VEL
LIN {X 0,Y 365.47,Z 621.989,A -85,B 0,C 180,E1 14255.443,E2 14255.443} C_VEL
LIN {X 0,Y 366.291,Z 621.054,A -85,B 0,C 180,E1 14257.55,E2 14257.55} C_VEL
LIN {X 0,Y 366.512,Z 629.133,A -85,B 0,C 180,E1 14259.72,E2 14259.72} C_VEL
LIN {X 0,Y 367.205,Z 646.78,A -85,B 0,C 180,E1 14262.474,E2 14262.474} C_VEL
LIN {X 0,Y 355.652,Z 690.146,A -85,B 0,C 180,E1 14265.803,E2 14265.803} C_VEL
LIN {X 0,Y 344.804,Z 729.342,A -85,B 0,C 180,E1 14270.05,E2 14270.05} C_VEL
LIN {X 0,Y 335.067,Z 763.837,A -85,B 0,C 180,E1 14275.215,E2 14275.215} C_VEL
LIN {X 0,Y 327.536,Z 791.853,A -85,B 0,C 180,E1 14280.971,E2 14280.971} C_VEL
LIN {X 0,Y 322.205,Z 814.455,A -85,B 0,C 180,E1 14287.361,E2 14287.361} C_VEL
LIN {X 0,Y 319.55,Z 829.987,A -85,B 0,C 180,E1 14293.483,E2 14293.483} C_VEL
LIN {X 0,Y 318.379,Z 841.445,A -85,B 0,C 180,E1 14300.418,E2 14300.418} C_VEL
LIN {X 0,Y 318.262,Z 846.95,A -85,B 0,C 180,E1 14307.319,E2 14307.319} C_VEL
LIN {X 0,Y 318.273,Z 847.131,A -85,B 0,C 180,E1 14312.725,E2 14312.725} C_VEL
LIN {X 0,Y 318.236,Z 843.697,A -85,B 0,C 180,E1 14318.205,E2 14318.205} C_VEL
LIN {X 0,Y 319.038,Z 835.378,A -85,B 0,C 180,E1 14324.426,E2 14324.426} C_VEL
LIN {X 0,Y 321.244,Z 821.976,A -85,B 0,C 180,E1 14330.699,E2 14330.699} C_VEL
LIN {X 0,Y 323.438,Z 811.95,A -85,B 0,C 180,E1 14334.22,E2 14334.22} C_VEL
LIN {X 0,Y 321.625,Z 803.547,A -85,B 0,C 180,E1 14336.94,E2 14336.94} C_VEL
LIN {X 0,Y 320.368,Z 794.148,A -85,B 0,C 180,E1 14339.578,E2 14339.578} C_VEL
LIN {X 0,Y 328.021,Z 767.64,A -85,B 0,C 180,E1 14345.236,E2 14345.236} C_VEL
LIN {X 0,Y 336.838,Z 737.245,A -85,B 0,C 180,E1 14349.968,E2 14349.968} C_VEL
LIN {X 0,Y 346.344,Z 701.9,A -85,B 0,C 180,E1 14353.926,E2 14353.926} C_VEL
LIN {X 0,Y 354.951,Z 664.125,A -85,B 0,C 180,E1 14356.882,E2 14356.882} C_VEL
LIN {X 0,Y 357.809,Z 648.698,A -85,B 0,C 180,E1 14357.806,E2 14357.806} C_VEL
LIN {X 0,Y 343.274,Z 613.951,A -85,B 0,C 180,E1 14362.175,E2 14362.175} C_VEL
LIN {X 0,Y 323.858,Z 577.587,A -85,B 0,C 180,E1 14367.242,E2 14367.242} C_VEL
LIN {X 0,Y 308.029,Z 550.446,A -85,B 0,C 180,E1 14371.664,E2 14371.664} C_VEL
LIN {X 0,Y 307.945,Z 549.53,A -85,B 0,C 180,E1 14372.249,E2 14372.249} C_VEL
LIN {X 0,Y 308.312,Z 549.53,A -85,B 0,C 180,E1 14379.901,E2 14379.901} C_VEL
LIN {X 0,Y 308.678,Z 549.53,A -85,B 0,C 180,E1 14385.81,E2 14385.81} C_VEL
LIN {X 0,Y 309.281,Z 549.53,A -85,B 0,C 180,E1 14394.387,E2 14394.387} C_VEL
LIN {X 0,Y 309.707,Z 549.53,A -85,B 0,C 180,E1 14400.006,E2 14400.006} C_VEL
LIN {X 0,Y 309.3,Z 549.53,A -85,B 0,C 180,E1 14405.624,E2 14405.624} C_VEL
LIN {X 0,Y 308.665,Z 549.53,A -85,B 0,C 180,E1 14414.203,E2 14414.203} C_VEL
LIN {X 0,Y 308.237,Z 549.53,A -85,B 0,C 180,E1 14421.051,E2 14421.051} C_VEL
LIN {X 0,Y 307.885,Z 549.53,A -85,B 0,C 180,E1 14429.462,E2 14429.462} C_VEL
LIN {X 0,Y 307.572,Z 549.53,A -85,B 0,C 180,E1 14438.038,E2 14438.038} C_VEL
LIN {X 0,Y 307.563,Z 549.53,A -85,B 0,C 180,E1 14443.573,E2 14443.573} C_VEL
LIN {X 0,Y 307.603,Z 549.53,A -85,B 0,C 180,E1 14450.219,E2 14450.219} C_VEL
LIN {X 0,Y 307.713,Z 549.53,A -85,B 0,C 180,E1 14457.233,E2 14457.233} C_VEL
LIN {X 0,Y 308.003,Z 549.53,A -85,B 0,C 180,E1 14463.743,E2 14463.743} C_VEL
LIN {X 0,Y 308.342,Z 549.53,A -85,B 0,C 180,E1 14469.897,E2 14469.897} C_VEL
LIN {X 0,Y 308.704,Z 549.53,A -85,B 0,C 180,E1 14475.806,E2 14475.806} C_VEL
LIN {X 0,Y 309.355,Z 549.53,A -85,B 0,C 180,E1 14484.384,E2 14484.384} C_VEL
LIN {X 0,Y 309.8,Z 549.53,A -85,B 0,C 180,E1 14490.001,E2 14490.001} C_VEL
LIN {X 0,Y 309.1,Z 549.53,A -85,B 0,C 180,E1 14498.451,E2 14498.451} C_VEL
LIN {X 0,Y 308.613,Z 549.889,A -85,B 0,C 180,E1 14505.564,E2 14505.564} C_VEL
LIN {X 0,Y 314.242,Z 560.938,A -85,B 0,C 180,E1 14507.412,E2 14507.412} C_VEL
LIN {X 0,Y 329.947,Z 593.021,A -85,B 0,C 180,E1 14512.765,E2 14512.765} C_VEL
LIN {X 0,Y 341.55,Z 623.767,A -85,B 0,C 180,E1 14517.598,E2 14517.598} C_VEL
LIN {X 0,Y 348.216,Z 649.743,A -85,B 0,C 180,E1 14521.623,E2 14521.623} C_VEL
LIN {X 0,Y 339.216,Z 683.698,A -85,B 0,C 180,E1 14525.587,E2 14525.587} C_VEL
LIN {X 0,Y 329.947,Z 714.855,A -85,B 0,C 180,E1 14530.658,E2 14530.658} C_VEL
LIN {X 0,Y 321.861,Z 740.554,A -85,B 0,C 180,E1 14536.516,E2 14536.516} C_VEL
LIN {X 0,Y 316.056,Z 760.245,A -85,B 0,C 180,E1 14542.831,E2 14542.831} C_VEL
LIN {X 0,Y 312.526,Z 774.448,A -85,B 0,C 180,E1 14549.42,E2 14549.42} C_VEL
LIN {X 0,Y 310.861,Z 783.028,A -85,B 0,C 180,E1 14555.538,E2 14555.538} C_VEL
LIN {X 0,Y 309.85,Z 788.142,A -85,B 0,C 180,E1 14562.946,E2 14562.946} C_VEL
LIN {X 0,Y 310.099,Z 788.232,A -85,B 0,C 180,E1 14568.732,E2 14568.732} C_VEL
LIN {X 0,Y 311.442,Z 784.312,A -85,B 0,C 180,E1 14575.362,E2 14575.362} C_VEL
LIN {X 0,Y 314.222,Z 774.645,A -85,B 0,C 180,E1 14582.756,E2 14582.756} C_VEL
LIN {X 0,Y 319.292,Z 760.092,A -85,B 0,C 180,E1 14589.547,E2 14589.547} C_VEL
LIN {X 0,Y 326.89,Z 740.529,A -85,B 0,C 180,E1 14595.784,E2 14595.784} C_VEL
LIN {X 0,Y 336.668,Z 715.615,A -85,B 0,C 180,E1 14601.426,E2 14601.426} C_VEL
LIN {X 0,Y 347.759,Z 685.727,A -85,B 0,C 180,E1 14606.281,E2 14606.281} C_VEL
LIN {X 0,Y 358.384,Z 653.743,A -85,B 0,C 180,E1 14610.198,E2 14610.198} C_VEL
LIN {X 0,Y 360.921,Z 633.859,A -85,B 0,C 180,E1 14614.254,E2 14614.254} C_VEL
LIN {X 0,Y 362.246,Z 628.902,A -85,B 0,C 180,E1 14615.806,E2 14615.806} C_VEL
LIN {X 0,Y 362.976,Z 628.839,A -85,B 0,C 180,E1 14617.575,E2 14617.575} C_VEL
LIN {X 0,Y 362.51,Z 639.324,A -85,B 0,C 180,E1 14619.992,E2 14619.992} C_VEL
LIN {X 0,Y 361.87,Z 650.806,A -85,B 0,C 180,E1 14621.664,E2 14621.664} C_VEL
LIN {X 0,Y 349.192,Z 694.107,A -85,B 0,C 180,E1 14625.202,E2 14625.202} C_VEL
LIN {X 0,Y 337.393,Z 733.162,A -85,B 0,C 180,E1 14629.709,E2 14629.709} C_VEL
LIN {X 0,Y 327.203,Z 766.829,A -85,B 0,C 180,E1 14635.065,E2 14635.065} C_VEL
LIN {X 0,Y 319.654,Z 793.666,A -85,B 0,C 180,E1 14640.919,E2 14640.919} C_VEL
LIN {X 0,Y 314.283,Z 815.198,A -85,B 0,C 180,E1 14647.33,E2 14647.33} C_VEL
LIN {X 0,Y 311.565,Z 830.557,A -85,B 0,C 180,E1 14653.773,E2 14653.773} C_VEL
LIN {X 0,Y 310.51,Z 840.662,A -85,B 0,C 180,E1 14660.172,E2 14660.172} C_VEL
LIN {X 0,Y 310.394,Z 846.172,A -85,B 0,C 180,E1 14667.203,E2 14667.203} C_VEL
LIN {X 0,Y 310.413,Z 846.354,A -85,B 0,C 180,E1 14672.795,E2 14672.795} C_VEL
LIN {X 0,Y 310.365,Z 842.88,A -85,B 0,C 180,E1 14678.414,E2 14678.414} C_VEL
LIN {X 0,Y 311.22,Z 834.465,A -85,B 0,C 180,E1 14684.797,E2 14684.797} C_VEL
LIN {X 0,Y 313.591,Z 820.935,A -85,B 0,C 180,E1 14691.229,E2 14691.229} C_VEL
LIN {X 0,Y 318.334,Z 801.527,A -85,B 0,C 180,E1 14697.627,E2 14697.627} C_VEL
LIN {X 0,Y 320.368,Z 794.148,A -85,B 0,C 180,E1 14699.578,E2 14699.578} C_VEL
LIN {X 0,Y 319.497,Z 784.163,A -85,B 0,C 180,E1 14702.153,E2 14702.153} C_VEL
LIN {X 0,Y 318.962,Z 773.501,A -85,B 0,C 180,E1 14704.665,E2 14704.665} C_VEL
LIN {X 0,Y 328.489,Z 742.157,A -85,B 0,C 180,E1 14709.97,E2 14709.97} C_VEL
LIN {X 0,Y 338.712,Z 706.12,A -85,B 0,C 180,E1 14714.246,E2 14714.246} C_VEL
LIN {X 0,Y 347.547,Z 669.211,A -85,B 0,C 180,E1 14717.318,E2 14717.318} C_VEL
LIN {X 0,Y 350.948,Z 650.642,A -85,B 0,C 180,E1 14718.529,E2 14718.529} C_VEL
LIN {X 0,Y 337.204,Z 617.301,A -85,B 0,C 180,E1 14722.898,E2 14722.898} C_VEL
LIN {X 0,Y 317.414,Z 579.807,A -85,B 0,C 180,E1 14728.36,E2 14728.36} C_VEL
LIN {X 0,Y 301.667,Z 554.316,A -85,B 0,C 180,E1 14732.868,E2 14732.868} C_VEL
LIN {X 0,Y 300.109,Z 549.53,A -85,B 0,C 180,E1 14733.606,E2 14733.606} C_VEL
LIN {X 0,Y 300.534,Z 549.53,A -85,B 0,C 180,E1 14742.413,E2 14742.413} C_VEL
LIN {X 0,Y 300.951,Z 549.53,A -85,B 0,C 180,E1 14748.397,E2 14748.397} C_VEL
LIN {X 0,Y 301.643,Z 549.53,A -85,B 0,C 180,E1 14757.129,E2 14757.129} C_VEL
LIN {X 0,Y 301.69,Z 549.53,A -85,B 0,C 180,E1 14762.883,E2 14762.883} C_VEL
LIN {X 0,Y 300.918,Z 549.53,A -85,B 0,C 180,E1 14771.616,E2 14771.616} C_VEL
LIN {X 0,Y 300.557,Z 549.53,A -85,B 0,C 180,E1 14777.599,E2 14777.599} C_VEL
LIN {X 0,Y 300.099,Z 549.53,A -85,B 0,C 180,E1 14784.753,E2 14784.753} C_VEL
LIN {X 0,Y 299.794,Z 549.53,A -85,B 0,C 180,E1 14790.847,E2 14790.847} C_VEL
LIN {X 0,Y 299.67,Z 549.53,A -85,B 0,C 180,E1 14797.328,E2 14797.328} C_VEL
LIN {X 0,Y 299.573,Z 549.53,A -85,B 0,C 180,E1 14805.045,E2 14805.045} C_VEL
LIN {X 0,Y 299.667,Z 549.53,A -85,B 0,C 180,E1 14812.679,E2 14812.679} C_VEL
LIN {X 0,Y 299.844,Z 549.53,A -85,B 0,C 180,E1 14819.673,E2 14819.673} C_VEL
LIN {X 0,Y 300.146,Z 549.53,A -85,B 0,C 180,E1 14826.201,E2 14826.201} C_VEL
LIN {X 0,Y 300.673,Z 549.53,A -85,B 0,C 180,E1 14833.106,E2 14833.106} C_VEL
LIN {X 0,Y 301.142,Z 549.53,A -85,B 0,C 180,E1 14841.326,E2 14841.326} C_VEL
LIN {X 0,Y 301.719,Z 549.53,A -85,B 0,C 180,E1 14847.125,E2 14847.125} C_VEL
LIN {X 0,Y 301.716,Z 549.53,A -85,B 0,C 180,E1 14852.878,E2 14852.878} C_VEL
LIN {X 0,Y 300.944,Z 549.53,A -85,B 0,C 180,E1 14861.611,E2 14861.611} C_VEL
LIN {X 0,Y 300.79,Z 549.53,A -85,B 0,C 180,E1 14863.835,E2 14863.835} C_VEL
LIN {X 0,Y 303.161,Z 555.211,A -85,B 0,C 180,E1 14864.739,E2 14864.739} C_VEL
LIN {X 0,Y 318.892,Z 585.521,A -85,B 0,C 180,E1 14870.176,E2 14870.176} C_VEL
LIN {X 0,Y 330.955,Z 614.812,A -85,B 0,C 180,E1 14875.036,E2 14875.036} C_VEL
LIN {X 0,Y 339.757,Z 643.505,A -85,B 0,C 180,E1 14879.67,E2 14879.67} C_VEL
LIN {X 0,Y 341.231,Z 652.903,A -85,B 0,C 180,E1 14881.113,E2 14881.113} C_VEL
LIN {X 0,Y 331.366,Z 688.256,A -85,B 0,C 180,E1 14885.42,E2 14885.42} C_VEL
LIN {X 0,Y 322.211,Z 717.605,A -85,B 0,C 180,E1 14890.449,E2 14890.449} C_VEL
LIN {X 0,Y 314.16,Z 742.318,A -85,B 0,C 180,E1 14896.297,E2 14896.297} C_VEL
LIN {X 0,Y 308.263,Z 761.603,A -85,B 0,C 180,E1 14902.696,E2 14902.696} C_VEL
LIN {X 0,Y 304.645,Z 775.69,A -85,B 0,C 180,E1 14909.483,E2 14909.483} C_VEL
LIN {X 0,Y 302.809,Z 784.712,A -85,B 0,C 180,E1 14916.416,E2 14916.416} C_VEL
LIN {X 0,Y 301.994,Z 788.709,A -85,B 0,C 180,E1 14922.488,E2 14922.488} C_VEL
LIN {X 0,Y 302.189,Z 789.158,A -85,B 0,C 180,E1 14928.433,E2 14928.433} C_VEL
LIN {X 0,Y 303.693,Z 785.225,A -85,B 0,C 180,E1 14935.654,E2 14935.654} C_VEL
LIN {X 0,Y 306.456,Z 776.358,A -85,B 0,C 180,E1 14942.826,E2 14942.826} C_VEL
LIN {X 0,Y 311.757,Z 762.265,A -85,B 0,C 180,E1 14949.78,E2 14949.78} C_VEL
LIN {X 0,Y 319.658,Z 743.264,A -85,B 0,C 180,E1 14956.151,E2 14956.151} C_VEL
LIN {X 0,Y 329.837,Z 719.104,A -85,B 0,C 180,E1 14961.892,E2 14961.892} C_VEL
LIN {X 0,Y 342.32,Z 688.257,A -85,B 0,C 180,E1 14967.13,E2 14967.13} C_VEL
LIN {X 0,Y 353.581,Z 658.152,A -85,B 0,C 180,E1 14970.914,E2 14970.914} C_VEL
LIN {X 0,Y 357.775,Z 638.825,A -85,B 0,C 180,E1 14975.156,E2 14975.156} C_VEL
LIN {X 0,Y 358.967,Z 636.008,A -85,B 0,C 180,E1 14976.185,E2 14976.185} C_VEL
LIN {X 0,Y 359.55,Z 636.014,A -85,B 0,C 180,E1 14977.332,E2 14977.332} C_VEL
LIN {X 0,Y 358.005,Z 648.237,A -85,B 0,C 180,E1 14979.974,E2 14979.974} C_VEL
LIN {X 0,Y 357.017,Z 654.405,A -85,B 0,C 180,E1 14980.77,E2 14980.77} C_VEL
LIN {X 0,Y 342.75,Z 698.042,A -85,B 0,C 180,E1 14984.576,E2 14984.576} C_VEL
LIN {X 0,Y 330.254,Z 736.318,A -85,B 0,C 180,E1 14989.253,E2 14989.253} C_VEL
LIN {X 0,Y 319.326,Z 770.077,A -85,B 0,C 180,E1 14994.95,E2 14994.95} C_VEL
LIN {X 0,Y 311.376,Z 796.726,A -85,B 0,C 180,E1 15001.177,E2 15001.177} C_VEL
LIN {X 0,Y 305.948,Z 818.333,A -85,B 0,C 180,E1 15008.212,E2 15008.212} C_VEL
LIN {X 0,Y 303.194,Z 833.691,A -85,B 0,C 180,E1 15015.54,E2 15015.54} C_VEL
LIN {X 0,Y 302.533,Z 841.415,A -85,B 0,C 180,E1 15021.364,E2 15021.364} C_VEL
LIN {X 0,Y 302.511,Z 845.409,A -85,B 0,C 180,E1 15027.13,E2 15027.13} C_VEL
LIN {X 0,Y 302.531,Z 845.57,A -85,B 0,C 180,E1 15032.867,E2 15032.867} C_VEL
LIN {X 0,Y 302.518,Z 842.063,A -85,B 0,C 180,E1 15038.634,E2 15038.634} C_VEL
LIN {X 0,Y 303.429,Z 833.553,A -85,B 0,C 180,E1 15045.186,E2 15045.186} C_VEL
LIN {X 0,Y 305.982,Z 819.867,A -85,B 0,C 180,E1 15051.783,E2 15051.783} C_VEL
LIN {X 0,Y 311.01,Z 800.223,A -85,B 0,C 180,E1 15058.335,E2 15058.335} C_VEL
LIN {X 0,Y 318.204,Z 776.035,A -85,B 0,C 180,E1 15064.15,E2 15064.15} C_VEL
LIN {X 0,Y 318.962,Z 773.501,A -85,B 0,C 180,E1 15064.665,E2 15064.665} C_VEL
LIN {X 0,Y 318.864,Z 762.263,A -85,B 0,C 180,E1 15067.088,E2 15067.088} C_VEL
LIN {X 0,Y 319.059,Z 750.286,A -85,B 0,C 180,E1 15069.392,E2 15069.392} C_VEL
LIN {X 0,Y 329.216,Z 716.439,A -85,B 0,C 180,E1 15073.895,E2 15073.895} C_VEL
LIN {X 0,Y 338.824,Z 679.509,A -85,B 0,C 180,E1 15077.367,E2 15077.367} C_VEL
LIN {X 0,Y 344.37,Z 653.404,A -85,B 0,C 180,E1 15079.166,E2 15079.166} C_VEL
LIN {X 0,Y 330.441,Z 619.237,A -85,B 0,C 180,E1 15083.856,E2 15083.856} C_VEL
LIN {X 0,Y 311.573,Z 583.086,A -85,B 0,C 180,E1 15089.328,E2 15089.328} C_VEL
LIN {X 0,Y 293.975,Z 554.561,A -85,B 0,C 180,E1 15094.637,E2 15094.637} C_VEL
LIN {X 0,Y 292.185,Z 549.53,A -85,B 0,C 180,E1 15095.517,E2 15095.517} C_VEL
LIN {X 0,Y 292.542,Z 549.53,A -85,B 0,C 180,E1 15101.916,E2 15101.916} C_VEL
LIN {X 0,Y 293.02,Z 549.53,A -85,B 0,C 180,E1 15109.03,E2 15109.03} C_VEL
LIN {X 0,Y 293.719,Z 549.53,A -85,B 0,C 180,E1 15117.051,E2 15117.051} C_VEL
LIN {X 0,Y 293.764,Z 549.53,A -85,B 0,C 180,E1 15122.96,E2 15122.96} C_VEL
LIN {X 0,Y 292.983,Z 549.53,A -85,B 0,C 180,E1 15131.936,E2 15131.936} C_VEL
LIN {X 0,Y 292.567,Z 549.53,A -85,B 0,C 180,E1 15138.096,E2 15138.096} C_VEL
LIN {X 0,Y 292.213,Z 549.53,A -85,B 0,C 180,E1 15144.495,E2 15144.495} C_VEL
LIN {X 0,Y 291.864,Z 549.53,A -85,B 0,C 180,E1 15151.255,E2 15151.255} C_VEL
LIN {X 0,Y 291.627,Z 549.53,A -85,B 0,C 180,E1 15158.854,E2 15158.854} C_VEL
LIN {X 0,Y 291.547,Z 549.53,A -85,B 0,C 180,E1 15167.538,E2 15167.538} C_VEL
LIN {X 0,Y 291.82,Z 549.53,A -85,B 0,C 180,E1 15176.122,E2 15176.122} C_VEL
LIN {X 0,Y 292.01,Z 549.53,A -85,B 0,C 180,E1 15182.185,E2 15182.185} C_VEL
LIN {X 0,Y 292.365,Z 549.53,A -85,B 0,C 180,E1 15188.788,E2 15188.788} C_VEL
LIN {X 0,Y 292.815,Z 549.53,A -85,B 0,C 180,E1 15195.018,E2 15195.018} C_VEL
LIN {X 0,Y 293.196,Z 549.53,A -85,B 0,C 180,E1 15201.089,E2 15201.089} C_VEL
LIN {X 0,Y 293.794,Z 549.53,A -85,B 0,C 180,E1 15207.047,E2 15207.047} C_VEL
LIN {X 0,Y 293.79,Z 549.53,A -85,B 0,C 180,E1 15212.955,E2 15212.955} C_VEL
LIN {X 0,Y 292.986,Z 549.53,A -85,B 0,C 180,E1 15222.035,E2 15222.035} C_VEL
LIN {X 0,Y 295.227,Z 555.087,A -85,B 0,C 180,E1 15222.969,E2 15222.969} C_VEL
LIN {X 0,Y 310.562,Z 583.954,A -85,B 0,C 180,E1 15228.476,E2 15228.476} C_VEL
LIN {X 0,Y 323.446,Z 614.83,A -85,B 0,C 180,E1 15233.813,E2 15233.813} C_VEL
LIN {X 0,Y 332.653,Z 644.795,A -85,B 0,C 180,E1 15238.827,E2 15238.827} C_VEL
LIN {X 0,Y 334.586,Z 654.559,A -85,B 0,C 180,E1 15240.441,E2 15240.441} C_VEL
LIN {X 0,Y 324.39,Z 689.674,A -85,B 0,C 180,E1 15244.818,E2 15244.818} C_VEL
LIN {X 0,Y 315.237,Z 718.14,A -85,B 0,C 180,E1 15249.776,E2 15249.776} C_VEL
LIN {X 0,Y 306.933,Z 742.658,A -85,B 0,C 180,E1 15255.658,E2 15255.658} C_VEL
LIN {X 0,Y 300.71,Z 762.198,A -85,B 0,C 180,E1 15262.251,E2 15262.251} C_VEL
LIN {X 0,Y 296.863,Z 776.56,A -85,B 0,C 180,E1 15269.328,E2 15269.328} C_VEL
LIN {X 0,Y 295.063,Z 784.939,A -85,B 0,C 180,E1 15275.757,E2 15275.757} C_VEL
LIN {X 0,Y 294.163,Z 789.239,A -85,B 0,C 180,E1 15282.006,E2 15282.006} C_VEL
LIN {X 0,Y 294.296,Z 790.086,A -85,B 0,C 180,E1 15288.118,E2 15288.118} C_VEL
LIN {X 0,Y 295.824,Z 786.539,A -85,B 0,C 180,E1 15295.539,E2 15295.539} C_VEL
LIN {X 0,Y 298.695,Z 778.088,A -85,B 0,C 180,E1 15302.899,E2 15302.899} C_VEL
LIN {X 0,Y 304.24,Z 764.479,A -85,B 0,C 180,E1 15310.025,E2 15310.025} C_VEL
LIN {X 0,Y 312.985,Z 744.901,A -85,B 0,C 180,E1 15316.866,E2 15316.866} C_VEL
LIN {X 0,Y 324.428,Z 719.724,A -85,B 0,C 180,E1 15323.001,E2 15323.001} C_VEL
LIN {X 0,Y 337.759,Z 689.28,A -85,B 0,C 180,E1 15328.254,E2 15328.254} C_VEL
LIN {X 0,Y 349.179,Z 661.862,A -85,B 0,C 180,E1 15331.825,E2 15331.825} C_VEL
LIN {X 0,Y 354.591,Z 644.905,A -85,B 0,C 180,E1 15335.777,E2 15335.777} C_VEL
LIN {X 0,Y 355.627,Z 643.054,A -85,B 0,C 180,E1 15336.58,E2 15336.58} C_VEL
LIN {X 0,Y 355.415,Z 644.744,A -85,B 0,C 180,E1 15337.493,E2 15337.493} C_VEL
LIN {X 0,Y 352.949,Z 656.704,A -85,B 0,C 180,E1 15339.742,E2 15339.742} C_VEL
LIN {X 0,Y 337.363,Z 699.493,A -85,B 0,C 180,E1 15343.639,E2 15343.639} C_VEL
LIN {X 0,Y 323.422,Z 738.69,A -85,B 0,C 180,E1 15348.647,E2 15348.647} C_VEL
LIN {X 0,Y 311.76,Z 772.311,A -85,B 0,C 180,E1 15354.663,E2 15354.663} C_VEL
LIN {X 0,Y 303.578,Z 797.912,A -85,B 0,C 180,E1 15360.973,E2 15360.973} C_VEL
LIN {X 0,Y 298.302,Z 817.584,A -85,B 0,C 180,E1 15367.623,E2 15367.623} C_VEL
LIN {X 0,Y 295.627,Z 831.738,A -85,B 0,C 180,E1 15374.401,E2 15374.401} C_VEL
LIN {X 0,Y 294.654,Z 840.657,A -85,B 0,C 180,E1 15381.131,E2 15381.131} C_VEL
LIN {X 0,Y 294.65,Z 844.639,A -85,B 0,C 180,E1 15387.053,E2 15387.053} C_VEL
LIN {X 0,Y 294.67,Z 844.78,A -85,B 0,C 180,E1 15392.944,E2 15392.944} C_VEL
LIN {X 0,Y 294.645,Z 841.222,A -85,B 0,C 180,E1 15398.867,E2 15398.867} C_VEL
LIN {X 0,Y 295.638,Z 832.594,A -85,B 0,C 180,E1 15405.596,E2 15405.596} C_VEL
LIN {X 0,Y 298.359,Z 818.749,A -85,B 0,C 180,E1 15412.369,E2 15412.369} C_VEL
LIN {X 0,Y 303.746,Z 799.055,A -85,B 0,C 180,E1 15419.037,E2 15419.037} C_VEL
LIN {X 0,Y 311.498,Z 773.962,A -85,B 0,C 180,E1 15425.115,E2 15425.115} C_VEL
LIN {X 0,Y 319.059,Z 750.286,A -85,B 0,C 180,E1 15429.392,E2 15429.392} C_VEL
LIN {X 0,Y 319.484,Z 737.741,A -85,B 0,C 180,E1 15431.591,E2 15431.591} C_VEL
LIN {X 0,Y 320.058,Z 724.641,A -85,B 0,C 180,E1 15433.677,E2 15433.677} C_VEL
LIN {X 0,Y 330.146,Z 688.886,A -85,B 0,C 180,E1 15437.409,E2 15437.409} C_VEL
LIN {X 0,Y 337.603,Z 655.622,A -85,B 0,C 180,E1 15439.898,E2 15439.898} C_VEL
LIN {X 0,Y 324.989,Z 624.046,A -85,B 0,C 180,E1 15444.392,E2 15444.392} C_VEL
LIN {X 0,Y 307.28,Z 589.032,A -85,B 0,C 180,E1 15449.877,E2 15449.877} C_VEL
LIN {X 0,Y 287.003,Z 555.51,A -85,B 0,C 180,E1 15456.289,E2 15456.289} C_VEL
LIN {X 0,Y 284.304,Z 550.284,A -85,B 0,C 180,E1 15457.296,E2 15457.296} C_VEL
LIN {X 0,Y 284.796,Z 549.53,A -85,B 0,C 180,E1 15464.592,E2 15464.592} C_VEL
LIN {X 0,Y 285.23,Z 549.53,A -85,B 0,C 180,E1 15470.844,E2 15470.844} C_VEL
LIN {X 0,Y 285.817,Z 549.53,A -85,B 0,C 180,E1 15476.97,E2 15476.97} C_VEL
LIN {X 0,Y 285.856,Z 549.53,A -85,B 0,C 180,E1 15483.042,E2 15483.042} C_VEL
LIN {X 0,Y 285.016,Z 549.53,A -85,B 0,C 180,E1 15492.274,E2 15492.274} C_VEL
LIN {X 0,Y 284.586,Z 549.53,A -85,B 0,C 180,E1 15498.622,E2 15498.622} C_VEL
LIN {X 0,Y 284.199,Z 549.53,A -85,B 0,C 180,E1 15505.233,E2 15505.233} C_VEL
LIN {X 0,Y 283.877,Z 549.53,A -85,B 0,C 180,E1 15512.239,E2 15512.239} C_VEL
LIN {X 0,Y 283.592,Z 549.53,A -85,B 0,C 180,E1 15519.849,E2 15519.849} C_VEL
LIN {X 0,Y 283.561,Z 549.53,A -85,B 0,C 180,E1 15528.384,E2 15528.384} C_VEL
LIN {X 0,Y 283.694,Z 549.53,A -85,B 0,C 180,E1 15534.052,E2 15534.052} C_VEL
LIN {X 0,Y 284.02,Z 549.53,A -85,B 0,C 180,E1 15541.331,E2 15541.331} C_VEL
LIN {X 0,Y 284.362,Z 549.53,A -85,B 0,C 180,E1 15548.119,E2 15548.119} C_VEL
LIN {X 0,Y 284.827,Z 549.53,A -85,B 0,C 180,E1 15554.588,E2 15554.588} C_VEL
LIN {X 0,Y 285.259,Z 549.53,A -85,B 0,C 180,E1 15560.839,E2 15560.839} C_VEL
LIN {X 0,Y 285.887,Z 549.53,A -85,B 0,C 180,E1 15566.965,E2 15566.965} C_VEL
LIN {X 0,Y 285.883,Z 549.53,A -85,B 0,C 180,E1 15573.037,E2 15573.037} C_VEL
LIN {X 0,Y 285.197,Z 550.275,A -85,B 0,C 180,E1 15580.21,E2 15580.21} C_VEL
LIN {X 0,Y 288.154,Z 555.754,A -85,B 0,C 180,E1 15581.327,E2 15581.327} C_VEL
LIN {X 0,Y 304.003,Z 586.306,A -85,B 0,C 180,E1 15587.388,E2 15587.388} C_VEL
LIN {X 0,Y 315.965,Z 614.745,A -85,B 0,C 180,E1 15592.543,E2 15592.543} C_VEL
LIN {X 0,Y 325.502,Z 645.612,A -85,B 0,C 180,E1 15597.889,E2 15597.889} C_VEL
LIN {X 0,Y 327.443,Z 658.112,A -85,B 0,C 180,E1 15599.953,E2 15599.953} C_VEL
LIN {X 0,Y 317.018,Z 692.498,A -85,B 0,C 180,E1 15604.414,E2 15604.414} C_VEL
LIN {X 0,Y 307.278,Z 721.496,A -85,B 0,C 180,E1 15609.686,E2 15609.686} C_VEL
LIN {X 0,Y 299.083,Z 744.818,A -85,B 0,C 180,E1 15615.54,E2 15615.54} C_VEL
LIN {X 0,Y 292.763,Z 764.05,A -85,B 0,C 180,E1 15622.316,E2 15622.316} C_VEL
LIN {X 0,Y 288.949,Z 777.962,A -85,B 0,C 180,E1 15629.511,E2 15629.511} C_VEL
LIN {X 0,Y 286.98,Z 786.823,A -85,B 0,C 180,E1 15636.97,E2 15636.97} C_VEL
LIN {X 0,Y 286.197,Z 790.768,A -85,B 0,C 180,E1 15644.656,E2 15644.656} C_VEL
LIN {X 0,Y 287.026,Z 789.707,A -85,B 0,C 180,E1 15652.012,E2 15652.012} C_VEL
LIN {X 0,Y 288.908,Z 785.156,A -85,B 0,C 180,E1 15658.492,E2 15658.492} C_VEL
LIN {X 0,Y 292.925,Z 775.172,A -85,B 0,C 180,E1 15665.927,E2 15665.927} C_VEL
LIN {X 0,Y 299.908,Z 759.892,A -85,B 0,C 180,E1 15673.124,E2 15673.124} C_VEL
LIN {X 0,Y 310.422,Z 738.41,A -85,B 0,C 180,E1 15679.957,E2 15679.957} C_VEL
LIN {X 0,Y 323.733,Z 711.202,A -85,B 0,C 180,E1 15685.999,E2 15685.999} C_VEL
LIN {X 0,Y 339.667,Z 677.591,A -85,B 0,C 180,E1 15691.203,E2 15691.203} C_VEL
LIN {X 0,Y 345.294,Z 665.031,A -85,B 0,C 180,E1 15692.92,E2 15692.92} C_VEL
LIN {X 0,Y 351.712,Z 650.696,A -85,B 0,C 180,E1 15696.584,E2 15696.584} C_VEL
LIN {X 0,Y 350.723,Z 654.207,A -85,B 0,C 180,E1 15697.72,E2 15697.72} C_VEL
LIN {X 0,Y 349.194,Z 659.637,A -85,B 0,C 180,E1 15698.696,E2 15698.696} C_VEL
LIN {X 0,Y 331.625,Z 702.68,A -85,B 0,C 180,E1 15702.83,E2 15702.83} C_VEL
LIN {X 0,Y 316.305,Z 741.897,A -85,B 0,C 180,E1 15708.151,E2 15708.151} C_VEL
LIN {X 0,Y 304.041,Z 775.137,A -85,B 0,C 180,E1 15714.463,E2 15714.463} C_VEL
LIN {X 0,Y 295.281,Z 801.113,A -85,B 0,C 180,E1 15721.339,E2 15721.339} C_VEL
LIN {X 0,Y 289.623,Z 821.716,A -85,B 0,C 180,E1 15729.112,E2 15729.112} C_VEL
LIN {X 0,Y 287.188,Z 835.177,A -85,B 0,C 180,E1 15736.769,E2 15736.769} C_VEL
LIN {X 0,Y 286.693,Z 842.378,A -85,B 0,C 180,E1 15743.936,E2 15743.936} C_VEL
LIN {X 0,Y 286.984,Z 844.407,A -85,B 0,C 180,E1 15749.999,E2 15749.999} C_VEL
LIN {X 0,Y 286.724,Z 842.641,A -85,B 0,C 180,E1 15756.061,E2 15756.061} C_VEL
LIN {X 0,Y 287.265,Z 835.684,A -85,B 0,C 180,E1 15763.279,E2 15763.279} C_VEL
LIN {X 0,Y 289.363,Z 823.621,A -85,B 0,C 180,E1 15770.342,E2 15770.342} C_VEL
LIN {X 0,Y 294.34,Z 804.997,A -85,B 0,C 180,E1 15777.576,E2 15777.576} C_VEL
LIN {X 0,Y 301.935,Z 780.987,A -85,B 0,C 180,E1 15784.113,E2 15784.113} C_VEL
LIN {X 0,Y 311.602,Z 751.523,A -85,B 0,C 180,E1 15789.848,E2 15789.848} C_VEL
LIN {X 0,Y 320.058,Z 724.641,A -85,B 0,C 180,E1 15793.677,E2 15793.677} C_VEL
LIN {X 0,Y 320.756,Z 711.027,A -85,B 0,C 180,E1 15795.651,E2 15795.651} C_VEL
LIN {X 0,Y 321.564,Z 696.86,A -85,B 0,C 180,E1 15797.5,E2 15797.5} C_VEL
LIN {X 0,Y 330.925,Z 658.078,A -85,B 0,C 180,E1 15800.606,E2 15800.606} C_VEL
LIN {X 0,Y 318.597,Z 626.815,A -85,B 0,C 180,E1 15805.239,E2 15805.239} C_VEL
LIN {X 0,Y 301.096,Z 591.751,A -85,B 0,C 180,E1 15811.001,E2 15811.001} C_VEL
LIN {X 0,Y 282.655,Z 561.292,A -85,B 0,C 180,E1 15817.052,E2 15817.052} C_VEL
LIN {X 0,Y 276.472,Z 550.376,A -85,B 0,C 180,E1 15819.416,E2 15819.416} C_VEL
LIN {X 0,Y 276.556,Z 549.53,A -85,B 0,C 180,E1 15820.831,E2 15820.831} C_VEL
LIN {X 0,Y 277.063,Z 549.53,A -85,B 0,C 180,E1 15827.381,E2 15827.381} C_VEL
LIN {X 0,Y 277.888,Z 549.53,A -85,B 0,C 180,E1 15836.883,E2 15836.883} C_VEL
LIN {X 0,Y 277.926,Z 549.53,A -85,B 0,C 180,E1 15843.129,E2 15843.129} C_VEL
LIN {X 0,Y 277.052,Z 549.53,A -85,B 0,C 180,E1 15852.633,E2 15852.633} C_VEL
LIN {X 0,Y 276.455,Z 549.53,A -85,B 0,C 180,E1 15861.406,E2 15861.406} C_VEL
LIN {X 0,Y 276.046,Z 549.53,A -85,B 0,C 180,E1 15869.586,E2 15869.586} C_VEL
LIN {X 0,Y 275.695,Z 549.53,A -85,B 0,C 180,E1 15877.171,E2 15877.171} C_VEL
LIN {X 0,Y 275.624,Z 549.53,A -85,B 0,C 180,E1 15885.579,E2 15885.579} C_VEL
LIN {X 0,Y 275.694,Z 549.53,A -85,B 0,C 180,E1 15892.837,E2 15892.837} C_VEL
LIN {X 0,Y 276.146,Z 549.53,A -85,B 0,C 180,E1 15901.324,E2 15901.324} C_VEL
LIN {X 0,Y 276.45,Z 549.53,A -85,B 0,C 180,E1 15908.615,E2 15908.615} C_VEL
LIN {X 0,Y 277.093,Z 549.53,A -85,B 0,C 180,E1 15917.377,E2 15917.377} C_VEL
LIN {X 0,Y 277.958,Z 549.53,A -85,B 0,C 180,E1 15926.879,E2 15926.879} C_VEL
LIN {X 0,Y 277.953,Z 549.53,A -85,B 0,C 180,E1 15933.124,E2 15933.124} C_VEL
LIN {X 0,Y 277.397,Z 550.164,A -85,B 0,C 180,E1 15938.14,E2 15938.14} C_VEL
LIN {X 0,Y 280.015,Z 555.425,A -85,B 0,C 180,E1 15939.239,E2 15939.239} C_VEL
LIN {X 0,Y 295.381,Z 584.051,A -85,B 0,C 180,E1 15945.377,E2 15945.377} C_VEL
LIN {X 0,Y 308.258,Z 613.992,A -85,B 0,C 180,E1 15951.068,E2 15951.068} C_VEL
LIN {X 0,Y 317.774,Z 644.285,A -85,B 0,C 180,E1 15956.532,E2 15956.532} C_VEL
LIN {X 0,Y 320.859,Z 659.561,A -85,B 0,C 180,E1 15959.228,E2 15959.228} C_VEL
LIN {X 0,Y 310.409,Z 692.937,A -85,B 0,C 180,E1 15963.616,E2 15963.616} C_VEL
LIN {X 0,Y 300.783,Z 720.682,A -85,B 0,C 180,E1 15968.687,E2 15968.687} C_VEL
LIN {X 0,Y 292.262,Z 744.15,A -85,B 0,C 180,E1 15974.577,E2 15974.577} C_VEL
LIN {X 0,Y 285.682,Z 763.146,A -85,B 0,C 180,E1 15981.222,E2 15981.222} C_VEL
LIN {X 0,Y 281.43,Z 777.645,A -85,B 0,C 180,E1 15988.6,E2 15988.6} C_VEL
LIN {X 0,Y 279.314,Z 786.7,A -85,B 0,C 180,E1 15995.905,E2 15995.905} C_VEL
LIN {X 0,Y 278.491,Z 790.272,A -85,B 0,C 180,E1 16000.955,E2 16000.955} C_VEL
LIN {X 0,Y 278.573,Z 791.746,A -85,B 0,C 180,E1 16008.052,E2 16008.052} C_VEL
LIN {X 0,Y 280.054,Z 788.974,A -85,B 0,C 180,E1 16015.342,E2 16015.342} C_VEL
LIN {X 0,Y 283.169,Z 781.423,A -85,B 0,C 180,E1 16023.058,E2 16023.058} C_VEL
LIN {X 0,Y 289.203,Z 768.865,A -85,B 0,C 180,E1 16030.552,E2 16030.552} C_VEL
LIN {X 0,Y 299.306,Z 749.69,A -85,B 0,C 180,E1 16038.043,E2 16038.043} C_VEL
LIN {X 0,Y 312.652,Z 724.523,A -85,B 0,C 180,E1 16044.681,E2 16044.681} C_VEL
LIN {X 0,Y 328.994,Z 693.527,A -85,B 0,C 180,E1 16050.406,E2 16050.406} C_VEL
LIN {X 0,Y 341.19,Z 670.05,A -85,B 0,C 180,E1 16053.674,E2 16053.674} C_VEL
LIN {X 0,Y 347.47,Z 658.747,A -85,B 0,C 180,E1 16056.778,E2 16056.778} C_VEL
LIN {X 0,Y 345.65,Z 663.227,A -85,B 0,C 180,E1 16057.653,E2 16057.653} C_VEL
LIN {X 0,Y 325.957,Z 706.03,A -85,B 0,C 180,E1 16061.994,E2 16061.994} C_VEL
LIN {X 0,Y 309.16,Z 745.485,A -85,B 0,C 180,E1 16067.669,E2 16067.669} C_VEL
LIN {X 0,Y 296.647,Z 776.942,A -85,B 0,C 180,E1 16074.029,E2 16074.029} C_VEL
LIN {X 0,Y 287.476,Z 802.328,A -85,B 0,C 180,E1 16081.157,E2 16081.157} C_VEL
LIN {X 0,Y 281.765,Z 821.958,A -85,B 0,C 180,E1 16088.977,E2 16088.977} C_VEL
LIN {X 0,Y 279.434,Z 833.795,A -85,B 0,C 180,E1 16095.888,E2 16095.888} C_VEL
LIN {X 0,Y 278.862,Z 840.484,A -85,B 0,C 180,E1 16102.197,E2 16102.197} C_VEL
LIN {X 0,Y 278.904,Z 843.09,A -85,B 0,C 180,E1 16106.887,E2 16106.887} C_VEL
LIN {X 0,Y 278.928,Z 843.177,A -85,B 0,C 180,E1 16113.11,E2 16113.11} C_VEL
LIN {X 0,Y 278.903,Z 839.509,A -85,B 0,C 180,E1 16119.372,E2 16119.372} C_VEL
LIN {X 0,Y 280.071,Z 830.629,A -85,B 0,C 180,E1 16126.487,E2 16126.487} C_VEL
LIN {X 0,Y 283.21,Z 816.509,A -85,B 0,C 180,E1 16133.602,E2 16133.602} C_VEL
LIN {X 0,Y 289.069,Z 797.045,A -85,B 0,C 180,E1 16140.405,E2 16140.405} C_VEL
LIN {X 0,Y 297.641,Z 771.723,A -85,B 0,C 180,E1 16146.723,E2 16146.723} C_VEL
LIN {X 0,Y 308.012,Z 741.199,A -85,B 0,C 180,E1 16152.16,E2 16152.16} C_VEL
LIN {X 0,Y 319.288,Z 705.012,A -85,B 0,C 180,E1 16156.678,E2 16156.678} C_VEL
LIN {X 0,Y 321.564,Z 696.86,A -85,B 0,C 180,E1 16157.5,E2 16157.5} C_VEL
LIN {X 0,Y 322.369,Z 682.255,A -85,B 0,C 180,E1 16159.232,E2 16159.232} C_VEL
LIN {X 0,Y 322.717,Z 669.165,A -85,B 0,C 180,E1 16160.651,E2 16160.651} C_VEL
LIN {X 0,Y 323.16,Z 667.159,A -85,B 0,C 180,E1 16160.797,E2 16160.797} C_VEL
LIN {X 0,Y 324.182,Z 660.315,A -85,B 0,C 180,E1 16161.371,E2 16161.371} C_VEL
LIN {X 0,Y 311.637,Z 628.233,A -85,B 0,C 180,E1 16166.333,E2 16166.333} C_VEL
LIN {X 0,Y 295.108,Z 594.697,A -85,B 0,C 180,E1 16172.077,E2 16172.077} C_VEL
LIN {X 0,Y 275.526,Z 562.011,A -85,B 0,C 180,E1 16178.912,E2 16178.912} C_VEL
LIN {X 0,Y 268.828,Z 551.248,A -85,B 0,C 180,E1 16181.579,E2 16181.579} C_VEL
LIN {X 0,Y 268.652,Z 549.53,A -85,B 0,C 180,E1 16182.005,E2 16182.005} C_VEL
LIN {X 0,Y 269.346,Z 549.53,A -85,B 0,C 180,E1 16190.299,E2 16190.299} C_VEL
LIN {X 0,Y 269.968,Z 549.53,A -85,B 0,C 180,E1 16196.792,E2 16196.792} C_VEL
LIN {X 0,Y 270.003,Z 549.53,A -85,B 0,C 180,E1 16203.221,E2 16203.221} C_VEL
LIN {X 0,Y 269.356,Z 549.53,A -85,B 0,C 180,E1 16209.715,E2 16209.715} C_VEL
LIN {X 0,Y 268.784,Z 549.53,A -85,B 0,C 180,E1 16216.747,E2 16216.747} C_VEL
LIN {X 0,Y 268.256,Z 549.53,A -85,B 0,C 180,E1 16225.44,E2 16225.44} C_VEL
LIN {X 0,Y 267.841,Z 549.53,A -85,B 0,C 180,E1 16234.429,E2 16234.429} C_VEL
LIN {X 0,Y 267.658,Z 549.53,A -85,B 0,C 180,E1 16242.758,E2 16242.758} C_VEL
LIN {X 0,Y 267.728,Z 549.53,A -85,B 0,C 180,E1 16251.534,E2 16251.534} C_VEL
LIN {X 0,Y 267.972,Z 549.53,A -85,B 0,C 180,E1 16259.437,E2 16259.437} C_VEL
LIN {X 0,Y 268.357,Z 549.53,A -85,B 0,C 180,E1 16266.739,E2 16266.739} C_VEL
LIN {X 0,Y 268.863,Z 549.53,A -85,B 0,C 180,E1 16273.648,E2 16273.648} C_VEL
LIN {X 0,Y 269.375,Z 549.53,A -85,B 0,C 180,E1 16280.294,E2 16280.294} C_VEL
LIN {X 0,Y 270.034,Z 549.53,A -85,B 0,C 180,E1 16286.787,E2 16286.787} C_VEL
LIN {X 0,Y 270.03,Z 549.53,A -85,B 0,C 180,E1 16293.216,E2 16293.216} C_VEL
LIN {X 0,Y 269.682,Z 549.61,A -85,B 0,C 180,E1 16295.943,E2 16295.943} C_VEL
LIN {X 0,Y 271.907,Z 555.114,A -85,B 0,C 180,E1 16296.998,E2 16296.998} C_VEL
LIN {X 0,Y 286.21,Z 580.996,A -85,B 0,C 180,E1 16302.994,E2 16302.994} C_VEL
LIN {X 0,Y 299.057,Z 609.602,A -85,B 0,C 180,E1 16308.831,E2 16308.831} C_VEL
LIN {X 0,Y 308.766,Z 638.359,A -85,B 0,C 180,E1 16314.249,E2 16314.249} C_VEL
LIN {X 0,Y 313.955,Z 661.986,A -85,B 0,C 180,E1 16318.588,E2 16318.588} C_VEL
LIN {X 0,Y 303.107,Z 695.393,A -85,B 0,C 180,E1 16323.123,E2 16323.123} C_VEL
LIN {X 0,Y 292.715,Z 724.212,A -85,B 0,C 180,E1 16328.617,E2 16328.617} C_VEL
LIN {X 0,Y 283.389,Z 749.137,A -85,B 0,C 180,E1 16335.309,E2 16335.309} C_VEL
LIN {X 0,Y 276.547,Z 768.679,A -85,B 0,C 180,E1 16342.963,E2 16342.963} C_VEL
LIN {X 0,Y 273.021,Z 780.922,A -85,B 0,C 180,E1 16350.052,E2 16350.052} C_VEL
LIN {X 0,Y 271.237,Z 788.424,A -85,B 0,C 180,E1 16356.992,E2 16356.992} C_VEL
LIN {X 0,Y 270.436,Z 792.085,A -85,B 0,C 180,E1 16363.737,E2 16363.737} C_VEL
LIN {X 0,Y 271.05,Z 792.211,A -85,B 0,C 180,E1 16370.346,E2 16370.346} C_VEL
LIN {X 0,Y 273.088,Z 788.304,A -85,B 0,C 180,E1 16377.956,E2 16377.956} C_VEL
LIN {X 0,Y 277.572,Z 778.912,A -85,B 0,C 180,E1 16386.256,E2 16386.256} C_VEL
LIN {X 0,Y 286.17,Z 763.145,A -85,B 0,C 180,E1 16394.548,E2 16394.548} C_VEL
LIN {X 0,Y 298.646,Z 741.469,A -85,B 0,C 180,E1 16401.949,E2 16401.949} C_VEL
LIN {X 0,Y 315.527,Z 712.485,A -85,B 0,C 180,E1 16408.668,E2 16408.668} C_VEL
LIN {X 0,Y 336.275,Z 677.043,A -85,B 0,C 180,E1 16414.243,E2 16414.243} C_VEL
LIN {X 0,Y 341.774,Z 668.08,A -85,B 0,C 180,E1 16416.301,E2 16416.301} C_VEL
LIN {X 0,Y 342.089,Z 667.85,A -85,B 0,C 180,E1 16416.658,E2 16416.658} C_VEL
LIN {X 0,Y 320.994,Z 708.574,A -85,B 0,C 180,E1 16421,E2 16421} C_VEL
LIN {X 0,Y 302.171,Z 748.666,A -85,B 0,C 180,E1 16427.113,E2 16427.113} C_VEL
LIN {X 0,Y 288.817,Z 779.911,A -85,B 0,C 180,E1 16433.859,E2 16433.859} C_VEL
LIN {X 0,Y 279.407,Z 804.455,A -85,B 0,C 180,E1 16441.253,E2 16441.253} C_VEL
LIN {X 0,Y 273.866,Z 822.46,A -85,B 0,C 180,E1 16448.94,E2 16448.94} C_VEL
LIN {X 0,Y 271.377,Z 835.081,A -85,B 0,C 180,E1 16457.103,E2 16457.103} C_VEL
LIN {X 0,Y 270.941,Z 840.88,A -85,B 0,C 180,E1 16463.582,E2 16463.582} C_VEL
LIN {X 0,Y 271.264,Z 842.831,A -85,B 0,C 180,E1 16469.999,E2 16469.999} C_VEL
LIN {X 0,Y 270.982,Z 840.97,A -85,B 0,C 180,E1 16476.415,E2 16476.415} C_VEL
LIN {X 0,Y 271.554,Z 834.217,A -85,B 0,C 180,E1 16483.706,E2 16483.706} C_VEL
LIN {X 0,Y 273.782,Z 822.66,A -85,B 0,C 180,E1 16490.896,E2 16490.896} C_VEL
LIN {X 0,Y 278.991,Z 804.676,A -85,B 0,C 180,E1 16498.348,E2 16498.348} C_VEL
LIN {X 0,Y 286.875,Z 781.649,A -85,B 0,C 180,E1 16505.025,E2 16505.025} C_VEL
LIN {X 0,Y 296.831,Z 753.558,A -85,B 0,C 180,E1 16510.849,E2 16510.849} C_VEL
LIN {X 0,Y 307.988,Z 720.572,A -85,B 0,C 180,E1 16515.714,E2 16515.714} C_VEL
LIN {X 0,Y 319.292,Z 682.073,A -85,B 0,C 180,E1 16519.658,E2 16519.658} C_VEL
LIN {X 0,Y 323.16,Z 667.159,A -85,B 0,C 180,E1 16520.797,E2 16520.797} C_VEL
LIN {X 0,Y 322.149,Z 661.678,A -85,B 0,C 180,E1 16521.53,E2 16521.53} C_VEL
LIN {X 0,Y 313.917,Z 652.517,A -85,B 0,C 180,E1 16523.708,E2 16523.708} C_VEL
LIN {X 0,Y 299.449,Z 618.239,A -85,B 0,C 180,E1 16529.447,E2 16529.447} C_VEL
LIN {X 0,Y 283.713,Z 588.263,A -85,B 0,C 180,E1 16535.112,E2 16535.112} C_VEL
LIN {X 0,Y 266.595,Z 560.553,A -85,B 0,C 180,E1 16541.592,E2 16541.592} C_VEL
LIN {X 0,Y 262.848,Z 554.731,A -85,B 0,C 180,E1 16543.166,E2 16543.166} C_VEL
LIN {X 0,Y 260.909,Z 549.53,A -85,B 0,C 180,E1 16544.439,E2 16544.439} C_VEL
LIN {X 0,Y 261.665,Z 549.53,A -85,B 0,C 180,E1 16553.362,E2 16553.362} C_VEL
LIN {X 0,Y 262.339,Z 549.53,A -85,B 0,C 180,E1 16560.007,E2 16560.007} C_VEL
LIN {X 0,Y 261.682,Z 549.53,A -85,B 0,C 180,E1 16566.652,E2 16566.652} C_VEL
LIN {X 0,Y 261.11,Z 549.53,A -85,B 0,C 180,E1 16573.418,E2 16573.418} C_VEL
LIN {X 0,Y 260.458,Z 549.53,A -85,B 0,C 180,E1 16581.555,E2 16581.555} C_VEL
LIN {X 0,Y 260.061,Z 549.53,A -85,B 0,C 180,E1 16589.159,E2 16589.159} C_VEL
LIN {X 0,Y 259.821,Z 549.53,A -85,B 0,C 180,E1 16595.651,E2 16595.651} C_VEL
LIN {X 0,Y 259.555,Z 549.53,A -85,B 0,C 180,E1 16604.435,E2 16604.435} C_VEL
LIN {X 0,Y 259.634,Z 549.53,A -85,B 0,C 180,E1 16610.1,E2 16610.1} C_VEL
LIN {X 0,Y 259.987,Z 549.53,A -85,B 0,C 180,E1 16618.392,E2 16618.392} C_VEL
LIN {X 0,Y 260.378,Z 549.53,A -85,B 0,C 180,E1 16625.983,E2 16625.983} C_VEL
LIN {X 0,Y 260.885,Z 549.53,A -85,B 0,C 180,E1 16633.133,E2 16633.133} C_VEL
LIN {X 0,Y 261.414,Z 549.53,A -85,B 0,C 180,E1 16639.995,E2 16639.995} C_VEL
LIN {X 0,Y 262.102,Z 549.53,A -85,B 0,C 180,E1 16646.69,E2 16646.69} C_VEL
LIN {X 0,Y 262.085,Z 549.53,A -85,B 0,C 180,E1 16653.521,E2 16653.521} C_VEL
LIN {X 0,Y 264.513,Z 555.41,A -85,B 0,C 180,E1 16654.824,E2 16654.824} C_VEL
LIN {X 0,Y 278.248,Z 580.135,A -85,B 0,C 180,E1 16660.979,E2 16660.979} C_VEL
LIN {X 0,Y 291.032,Z 608.112,A -85,B 0,C 180,E1 16667.017,E2 16667.017} C_VEL
LIN {X 0,Y 300.843,Z 636.39,A -85,B 0,C 180,E1 16672.567,E2 16672.567} C_VEL
LIN {X 0,Y 307.167,Z 662.613,A -85,B 0,C 180,E1 16677.633,E2 16677.633} C_VEL
LIN {X 0,Y 297.075,Z 694.337,A -85,B 0,C 180,E1 16682.039,E2 16682.039} C_VEL
LIN {X 0,Y 286.376,Z 723.164,A -85,B 0,C 180,E1 16687.52,E2 16687.52} C_VEL
LIN {X 0,Y 276.867,Z 747.529,A -85,B 0,C 180,E1 16694.008,E2 16694.008} C_VEL
LIN {X 0,Y 269.421,Z 767.86,A -85,B 0,C 180,E1 16701.81,E2 16701.81} C_VEL
LIN {X 0,Y 265.15,Z 781.867,A -85,B 0,C 180,E1 16710.016,E2 16710.016} C_VEL
LIN {X 0,Y 263.381,Z 789.126,A -85,B 0,C 180,E1 16716.897,E2 16716.897} C_VEL
LIN {X 0,Y 262.579,Z 792.712,A -85,B 0,C 180,E1 16723.237,E2 16723.237} C_VEL
LIN {X 0,Y 263.141,Z 793.175,A -85,B 0,C 180,E1 16730.053,E2 16730.053} C_VEL
LIN {X 0,Y 265.269,Z 789.705,A -85,B 0,C 180,E1 16737.895,E2 16737.895} C_VEL
LIN {X 0,Y 269.921,Z 780.825,A -85,B 0,C 180,E1 16746.434,E2 16746.434} C_VEL
LIN {X 0,Y 278.856,Z 765.698,A -85,B 0,C 180,E1 16754.939,E2 16754.939} C_VEL
LIN {X 0,Y 292.635,Z 743.823,A -85,B 0,C 180,E1 16762.825,E2 16762.825} C_VEL
LIN {X 0,Y 311.404,Z 714.466,A -85,B 0,C 180,E1 16769.884,E2 16769.884} C_VEL
LIN {X 0,Y 335.489,Z 677.87,A -85,B 0,C 180,E1 16775.915,E2 16775.915} C_VEL
LIN {X 0,Y 334.395,Z 679.837,A -85,B 0,C 180,E1 16776.32,E2 16776.32} C_VEL
LIN {X 0,Y 311.214,Z 720.589,A -85,B 0,C 180,E1 16781.259,E2 16781.259} C_VEL
LIN {X 0,Y 292.513,Z 757.698,A -85,B 0,C 180,E1 16787.708,E2 16787.708} C_VEL
LIN {X 0,Y 279.261,Z 786.68,A -85,B 0,C 180,E1 16794.765,E2 16794.765} C_VEL
LIN {X 0,Y 269.821,Z 810.303,A -85,B 0,C 180,E1 16802.874,E2 16802.874} C_VEL
LIN {X 0,Y 265.109,Z 826.258,A -85,B 0,C 180,E1 16810.839,E2 16810.839} C_VEL
LIN {X 0,Y 263.295,Z 836.644,A -85,B 0,C 180,E1 16818.893,E2 16818.893} C_VEL
LIN {X 0,Y 263.17,Z 841.541,A -85,B 0,C 180,E1 16826.7,E2 16826.7} C_VEL
LIN {X 0,Y 263.412,Z 842.041,A -85,B 0,C 180,E1 16829.999,E2 16829.999} C_VEL
LIN {X 0,Y 263.126,Z 840.116,A -85,B 0,C 180,E1 16836.607,E2 16836.607} C_VEL
LIN {X 0,Y 263.744,Z 833.23,A -85,B 0,C 180,E1 16844.12,E2 16844.12} C_VEL
LIN {X 0,Y 266.265,Z 821.153,A -85,B 0,C 180,E1 16851.69,E2 16851.69} C_VEL
LIN {X 0,Y 271.705,Z 803.235,A -85,B 0,C 180,E1 16859.181,E2 16859.181} C_VEL
LIN {X 0,Y 279.948,Z 780.25,A -85,B 0,C 180,E1 16865.928,E2 16865.928} C_VEL
LIN {X 0,Y 290.651,Z 751.269,A -85,B 0,C 180,E1 16871.97,E2 16871.97} C_VEL
LIN {X 0,Y 302.237,Z 718.094,A -85,B 0,C 180,E1 16876.844,E2 16876.844} C_VEL
LIN {X 0,Y 313.628,Z 679.886,A -85,B 0,C 180,E1 16880.719,E2 16880.719} C_VEL
LIN {X 0,Y 317.613,Z 663.226,A -85,B 0,C 180,E1 16882.032,E2 16882.032} C_VEL
LIN {X 0,Y 313.917,Z 652.517,A -85,B 0,C 180,E1 16883.708,E2 16883.708} C_VEL
LIN {X 0,Y 308.617,Z 644.655,A -85,B 0,C 180,E1 16885.384,E2 16885.384} C_VEL
LIN {X 0,Y 299.212,Z 634.258,A -85,B 0,C 180,E1 16888.051,E2 16888.051} C_VEL
LIN {X 0,Y 298.499,Z 632.776,A -85,B 0,C 180,E1 16888.333,E2 16888.333} C_VEL
LIN {X 0,Y 283.387,Z 601.332,A -85,B 0,C 180,E1 16894.229,E2 16894.229} C_VEL
LIN {X 0,Y 266.611,Z 572.69,A -85,B 0,C 180,E1 16900.734,E2 16900.734} C_VEL
LIN {X 0,Y 255.808,Z 555.478,A -85,B 0,C 180,E1 16905.439,E2 16905.439} C_VEL
LIN {X 0,Y 253.288,Z 550.504,A -85,B 0,C 180,E1 16906.724,E2 16906.724} C_VEL
LIN {X 0,Y 253.212,Z 549.53,A -85,B 0,C 180,E1 16907.05,E2 16907.05} C_VEL
LIN {X 0,Y 254.102,Z 549.53,A -85,B 0,C 180,E1 16916.591,E2 16916.591} C_VEL
LIN {X 0,Y 254.134,Z 549.53,A -85,B 0,C 180,E1 16923.423,E2 16923.423} C_VEL
LIN {X 0,Y 253.46,Z 549.53,A -85,B 0,C 180,E1 16930.331,E2 16930.331} C_VEL
LIN {X 0,Y 252.866,Z 549.53,A -85,B 0,C 180,E1 16937.427,E2 16937.427} C_VEL
LIN {X 0,Y 252.25,Z 549.53,A -85,B 0,C 180,E1 16945.801,E2 16945.801} C_VEL
LIN {X 0,Y 251.935,Z 549.53,A -85,B 0,C 180,E1 16952.751,E2 16952.751} C_VEL
LIN {X 0,Y 251.622,Z 549.53,A -85,B 0,C 180,E1 16961.453,E2 16961.453} C_VEL
LIN {X 0,Y 251.605,Z 549.53,A -85,B 0,C 180,E1 16968.554,E2 16968.554} C_VEL
LIN {X 0,Y 251.928,Z 549.53,A -85,B 0,C 180,E1 16977.298,E2 16977.298} C_VEL
LIN {X 0,Y 252.333,Z 549.53,A -85,B 0,C 180,E1 16985.166,E2 16985.166} C_VEL
LIN {X 0,Y 252.977,Z 549.53,A -85,B 0,C 180,E1 16993.275,E2 16993.275} C_VEL
LIN {X 0,Y 253.486,Z 549.53,A -85,B 0,C 180,E1 16999.679,E2 16999.679} C_VEL
LIN {X 0,Y 254.166,Z 549.53,A -85,B 0,C 180,E1 17006.586,E2 17006.586} C_VEL
LIN {X 0,Y 254.339,Z 550.055,A -85,B 0,C 180,E1 17011.068,E2 17011.068} C_VEL
LIN {X 0,Y 256.891,Z 555.462,A -85,B 0,C 180,E1 17012.424,E2 17012.424} C_VEL
LIN {X 0,Y 270.441,Z 579.465,A -85,B 0,C 180,E1 17018.858,E2 17018.858} C_VEL
LIN {X 0,Y 283.708,Z 608.445,A -85,B 0,C 180,E1 17025.477,E2 17025.477} C_VEL
LIN {X 0,Y 293.389,Z 636.143,A -85,B 0,C 180,E1 17031.178,E2 17031.178} C_VEL
LIN {X 0,Y 299.892,Z 662.615,A -85,B 0,C 180,E1 17036.476,E2 17036.476} C_VEL
LIN {X 0,Y 299.928,Z 667.777,A -85,B 0,C 180,E1 17037.36,E2 17037.36} C_VEL
LIN {X 0,Y 288.079,Z 701.54,A -85,B 0,C 180,E1 17042.305,E2 17042.305} C_VEL
LIN {X 0,Y 276.769,Z 730.335,A -85,B 0,C 180,E1 17048.318,E2 17048.318} C_VEL
LIN {X 0,Y 267.675,Z 753.184,A -85,B 0,C 180,E1 17055.089,E2 17055.089} C_VEL
LIN {X 0,Y 260.99,Z 770.951,A -85,B 0,C 180,E1 17062.606,E2 17062.606} C_VEL
LIN {X 0,Y 256.967,Z 783.953,A -85,B 0,C 180,E1 17070.909,E2 17070.909} C_VEL
LIN {X 0,Y 255.08,Z 791.441,A -85,B 0,C 180,E1 17079.13,E2 17079.13} C_VEL
LIN {X 0,Y 254.765,Z 794.139,A -85,B 0,C 180,E1 17086.241,E2 17086.241} C_VEL
LIN {X 0,Y 255.961,Z 793.328,A -85,B 0,C 180,E1 17093.199,E2 17093.199} C_VEL
LIN {X 0,Y 258.991,Z 788.123,A -85,B 0,C 180,E1 17101.668,E2 17101.668} C_VEL
LIN {X 0,Y 265.104,Z 778.179,A -85,B 0,C 180,E1 17109.858,E2 17109.858} C_VEL
LIN {X 0,Y 276.277,Z 761.451,A -85,B 0,C 180,E1 17118.36,E2 17118.36} C_VEL
LIN {X 0,Y 292.516,Z 738.058,A -85,B 0,C 180,E1 17126.094,E2 17126.094} C_VEL
LIN {X 0,Y 312.966,Z 709.274,A -85,B 0,C 180,E1 17132.554,E2 17132.554} C_VEL
LIN {X 0,Y 327.314,Z 689.842,A -85,B 0,C 180,E1 17135.727,E2 17135.727} C_VEL
LIN {X 0,Y 298.031,Z 737.467,A -85,B 0,C 180,E1 17142.553,E2 17142.553} C_VEL
LIN {X 0,Y 279.334,Z 772.719,A -85,B 0,C 180,E1 17149.933,E2 17149.933} C_VEL
LIN {X 0,Y 266.703,Z 799.698,A -85,B 0,C 180,E1 17158.059,E2 17158.059} C_VEL
LIN {X 0,Y 259.606,Z 818.033,A -85,B 0,C 180,E1 17165.903,E2 17165.903} C_VEL
LIN {X 0,Y 256.273,Z 830.64,A -85,B 0,C 180,E1 17173.701,E2 17173.701} C_VEL
LIN {X 0,Y 255.231,Z 838.277,A -85,B 0,C 180,E1 17181.47,E2 17181.47} C_VEL
LIN {X 0,Y 255.304,Z 840.772,A -85,B 0,C 180,E1 17186.599,E2 17186.599} C_VEL
LIN {X 0,Y 255.575,Z 841.244,A -85,B 0,C 180,E1 17189.999,E2 17189.999} C_VEL
LIN {X 0,Y 255.247,Z 839.253,A -85,B 0,C 180,E1 17196.812,E2 17196.812} C_VEL
LIN {X 0,Y 255.946,Z 832.22,A -85,B 0,C 180,E1 17204.56,E2 17204.56} C_VEL
